		//Переменные для работы с MPX_a2_2
	mpx_a2_2_in_v_1 	 		   		:WORD; //1-е Напрядение входа
	mpx_a2_2_in_v_2 	 		   		:WORD; //2-e Напряжение входа
	mpx_a2_2_in_v_3 	 		   		:WORD; //3-е Напряжение входа
	mpx_a2_2_in_freq 	 		   		:WORD; //Частота на входе
	mpx_a2_2_in_freq_real		   		:REAL; //Частота на входе (x0.1)
	mpx_a2_2_bypass_v_1  		   		:WORD; //1-е Напряжение байпаса
	mpx_a2_2_bypass_v_2  		   		:WORD; //2-е Напряжение байпаса
	mpx_a2_2_bypass_v_3  		   		:WORD; //3-е Напряжение байпаса
	mpx_a2_2_bypass_freq 		   		:WORD; //Частота байпаса
	mpx_a2_2_bypass_freq_real      		:REAL; //Частота байпаса
	mpx_a2_2_output_v_1  		   		:WORD; //1-е Напряжение выхода
	mpx_a2_2_output_v_2  		   		:WORD; //2-е Напряжение выхода
	mpx_a2_2_output_v_3  		   		:WORD; //3-е Напряжение выхода
	mpx_a2_2_output_i_1  		   		:WORD; //1-й Ток выхода
	mpx_a2_2_output_i_2  		   		:WORD; //2-й Ток выхода
	mpx_a2_2_output_i_3  		   		:WORD; //3-й Ток выхода
	mpx_a2_2_output_i_1_real       		:REAL; //1-й Ток выхода (x0.1)
	mpx_a2_2_output_i_2_real       		:REAL; //2-й Ток выхода (x0.1)
	mpx_a2_2_output_i_3_real       		:REAL; //3-й Ток выхода (x0.1)
	mpx_a2_2_output_active_power_1 		:WORD; //Активная мощность 1-й фазы
	mpx_a2_2_output_active_power_2 		:WORD; //Активная мощность 2-й фазы
	mpx_a2_2_output_active_power_3 		:WORD; //Активная мощность 3-й фазы
	mpx_a2_2_output_active_power_1_real :REAL; //Активная мощность 1-й фазы (x0.1)
	mpx_a2_2_output_active_power_2_real :REAL; //Активная мощность 2-й фазы (x0.1)
	mpx_a2_2_output_active_power_3_real :REAL; //Активная мощность 3-й фазы (x0.1)
	mpx_a2_2_output_freq 	       		:WORD; //Частота выхода
	mpx_a2_2_output_freq_real 	        :REAL; //Частота выхода (x0.1)
	mpx_a2_2_load_ph_1    	       		:WORD; //Загрузска 1-й фазы (%)
	mpx_a2_2_load_ph_2    		   		:WORD; //Загрузска 3-й фазы (%)
	mpx_a2_2_load_ph_3    	       		:WORD; //Загрузска 2-й фазы (%)
	mpx_a2_2_battery_voltage 	   		:WORD; //Напряжение батареи
	mpx_a2_2_battery_voltage_real  		:REAL; //Напряжение батареи (x0.1)
	mpx_a2_2_battery_current 	   		:WORD; //Ток батареи
	mpx_a2_2_battery_current_real  		:REAL; //Ток батареи (x0.1)
	mpx_a2_2_battery_capacity 	   		:WORD; //Остаточная емкость батареи (%)
	mpx_a2_2_battery_time 		   		:WORD; //Остаточное время автономии (минуты)
	mpx_a2_2_temp 				   		:WORD; //Температура
	mpx_a2_2_state_reg_1 	       		:WORD; //1-й Регистр состояния
	mpx_a2_2_state_1_as_bit 	   		:WORD_AS_BIT;
	mpx_a2_2_state_reg_2 		   		:WORD; //2-й Регистр состояния
	mpx_a2_2_state_2_as_bit 	   		:WORD_AS_BIT;
	mpx_a2_2_bypass_line_state 	   		:STRING; 
	mpx_a2_2_bypass_arrow_state    		:STRING;
	mpx_a2_2_battery_arrow_state 		:STRING; //состояние батареи
	mpx_a2_2_battery_line_state 		:STRING; //состояние батареи
	mpx_a2_2_input_state 		   		:STRING; //состояние входа
	mpx_a2_2_output_state 		   		:STRING; //состояние выхода
	mpx_a2_2_alarm                      :BOOL;
	
	//Переменные для работы с MPX_s1_1
	mpx_s1_1_in_v_1 	 		   		:WORD; //1-е Напрядение входа
	mpx_s1_1_in_v_2 	 		   		:WORD; //2-e Напряжение входа
	mpx_s1_1_in_v_3 	 		   		:WORD; //3-е Напряжение входа
	mpx_s1_1_in_freq 	 		   		:WORD; //Частота на входе
	mpx_s1_1_in_freq_real		   		:REAL; //Частота на входе (x0.1)
	mpx_s1_1_bypass_v_1  		   		:WORD; //1-е Напряжение байпаса
	mpx_s1_1_bypass_v_2  		   		:WORD; //2-е Напряжение байпаса
	mpx_s1_1_bypass_v_3  		   		:WORD; //3-е Напряжение байпаса
	mpx_s1_1_bypass_freq 		   		:WORD; //Частота байпаса
	mpx_s1_1_bypass_freq_real      		:REAL; //Частота байпаса
	mpx_s1_1_output_v_1  		   		:WORD; //1-е Напряжение выхода
	mpx_s1_1_output_v_2  		   		:WORD; //2-е Напряжение выхода
	mpx_s1_1_output_v_3  		   		:WORD; //3-е Напряжение выхода
	mpx_s1_1_output_i_1  		   		:WORD; //1-й Ток выхода
	mpx_s1_1_output_i_2  		   		:WORD; //2-й Ток выхода
	mpx_s1_1_output_i_3  		   		:WORD; //3-й Ток выхода
	mpx_s1_1_output_i_1_real       		:REAL; //1-й Ток выхода (x0.1)
	mpx_s1_1_output_i_2_real       		:REAL; //2-й Ток выхода (x0.1)
	mpx_s1_1_output_i_3_real       		:REAL; //3-й Ток выхода (x0.1)
	mpx_s1_1_output_active_power_1 		:WORD; //Активная мощность 1-й фазы
	mpx_s1_1_output_active_power_2 		:WORD; //Активная мощность 2-й фазы
	mpx_s1_1_output_active_power_3 		:WORD; //Активная мощность 3-й фазы
	mpx_s1_1_output_active_power_1_real :REAL; //Активная мощность 1-й фазы (x0.1)
	mpx_s1_1_output_active_power_2_real :REAL; //Активная мощность 2-й фазы (x0.1)
	mpx_s1_1_output_active_power_3_real :REAL; //Активная мощность 3-й фазы (x0.1)
	mpx_s1_1_output_freq 	       		:WORD; //Частота выхода
	mpx_s1_1_output_freq_real 	        :REAL; //Частота выхода (x0.1)
	mpx_s1_1_load_ph_1    	       		:WORD; //Загрузска 1-й фазы (%)
	mpx_s1_1_load_ph_2    		   		:WORD; //Загрузска 3-й фазы (%)
	mpx_s1_1_load_ph_3    	       		:WORD; //Загрузска 2-й фазы (%)
	mpx_s1_1_battery_voltage 	   		:WORD; //Напряжение батареи
	mpx_s1_1_battery_voltage_real  		:REAL; //Напряжение батареи (x0.1)
	mpx_s1_1_battery_current 	   		:WORD; //Ток батареи
	mpx_s1_1_battery_current_real  		:REAL; //Ток батареи (x0.1)
	mpx_s1_1_battery_capacity 	   		:WORD; //Остаточная емкость батареи (%)
	mpx_s1_1_battery_time 		   		:WORD; //Остаточное время автономии (минуты)
	mpx_s1_1_temp 				   		:WORD; //Температура
	mpx_s1_1_state_reg_1 	       		:WORD; //1-й Регистр состояния
	mpx_s1_1_state_1_as_bit 	   		:WORD_AS_BIT;
	mpx_s1_1_state_reg_2 		   		:WORD; //2-й Регистр состояния
	mpx_s1_1_state_2_as_bit 	   		:WORD_AS_BIT;
	mpx_s1_1_bypass_line_state 	   		:STRING; 
	mpx_s1_1_bypass_arrow_state    		:STRING;
	mpx_s1_1_battery_arrow_state 		:STRING; //состояние батареи
	mpx_s1_1_battery_line_state 		:STRING; //состояние батареи
	mpx_s1_1_input_state 		   		:STRING; //состояние входа
	mpx_s1_1_output_state 		   		:STRING; //состояние выхода
	mpx_s1_1_alarm                      :BOOL;
	
	//Переменные для работы с MPX_s1_2
	mpx_s1_2_in_v_1 	 		   		:WORD; //1-е Напрядение входа
	mpx_s1_2_in_v_2 	 		   		:WORD; //2-e Напряжение входа
	mpx_s1_2_in_v_3 	 		   		:WORD; //3-е Напряжение входа
	mpx_s1_2_in_freq 	 		   		:WORD; //Частота на входе
	mpx_s1_2_in_freq_real		   		:REAL; //Частота на входе (x0.1)
	mpx_s1_2_bypass_v_1  		   		:WORD; //1-е Напряжение байпаса
	mpx_s1_2_bypass_v_2  		   		:WORD; //2-е Напряжение байпаса
	mpx_s1_2_bypass_v_3  		   		:WORD; //3-е Напряжение байпаса
	mpx_s1_2_bypass_freq 		   		:WORD; //Частота байпаса
	mpx_s1_2_bypass_freq_real      		:REAL; //Частота байпаса
	mpx_s1_2_output_v_1  		   		:WORD; //1-е Напряжение выхода
	mpx_s1_2_output_v_2  		   		:WORD; //2-е Напряжение выхода
	mpx_s1_2_output_v_3  		   		:WORD; //3-е Напряжение выхода
	mpx_s1_2_output_i_1  		   		:WORD; //1-й Ток выхода
	mpx_s1_2_output_i_2  		   		:WORD; //2-й Ток выхода
	mpx_s1_2_output_i_3  		   		:WORD; //3-й Ток выхода
	mpx_s1_2_output_i_1_real       		:REAL; //1-й Ток выхода (x0.1)
	mpx_s1_2_output_i_2_real       		:REAL; //2-й Ток выхода (x0.1)
	mpx_s1_2_output_i_3_real       		:REAL; //3-й Ток выхода (x0.1)
	mpx_s1_2_output_active_power_1 		:WORD; //Активная мощность 1-й фазы
	mpx_s1_2_output_active_power_2 		:WORD; //Активная мощность 2-й фазы
	mpx_s1_2_output_active_power_3 		:WORD; //Активная мощность 3-й фазы
	mpx_s1_2_output_active_power_1_real :REAL; //Активная мощность 1-й фазы (x0.1)
	mpx_s1_2_output_active_power_2_real :REAL; //Активная мощность 2-й фазы (x0.1)
	mpx_s1_2_output_active_power_3_real :REAL; //Активная мощность 3-й фазы (x0.1)
	mpx_s1_2_output_freq 	       		:WORD; //Частота выхода
	mpx_s1_2_output_freq_real 	        :REAL; //Частота выхода (x0.1)
	mpx_s1_2_load_ph_1    	       		:WORD; //Загрузска 1-й фазы (%)
	mpx_s1_2_load_ph_2    		   		:WORD; //Загрузска 3-й фазы (%)
	mpx_s1_2_load_ph_3    	       		:WORD; //Загрузска 2-й фазы (%)
	mpx_s1_2_battery_voltage 	   		:WORD; //Напряжение батареи
	mpx_s1_2_battery_voltage_real  		:REAL; //Напряжение батареи (x0.1)
	mpx_s1_2_battery_current 	   		:WORD; //Ток батареи
	mpx_s1_2_battery_current_real  		:REAL; //Ток батареи (x0.1)
	mpx_s1_2_battery_capacity 	   		:WORD; //Остаточная емкость батареи (%)
	mpx_s1_2_battery_time 		   		:WORD; //Остаточное время автономии (минуты)
	mpx_s1_2_temp 				   		:WORD; //Температура
	mpx_s1_2_state_reg_1 	       		:WORD; //1-й Регистр состояния
	mpx_s1_2_state_1_as_bit 	   		:WORD_AS_BIT;
	mpx_s1_2_state_reg_2 		   		:WORD; //2-й Регистр состояния
	mpx_s1_2_state_2_as_bit 	   		:WORD_AS_BIT;
	mpx_s1_2_bypass_line_state 	   		:STRING; 
	mpx_s1_2_bypass_arrow_state    		:STRING;
	mpx_s1_2_battery_arrow_state 		:STRING; //состояние батареи
	mpx_s1_2_battery_line_state 		:STRING; //состояние батареи
	mpx_s1_2_input_state 		   		:STRING; //состояние входа
	mpx_s1_2_output_state 		   		:STRING; //состояние выхода
	mpx_s1_2_alarm                      :BOOL;
	
	//Переменные для работы с MPX_s1_3
	mpx_s1_3_in_v_1 	 		   		:WORD; //1-е Напрядение входа
	mpx_s1_3_in_v_2 	 		   		:WORD; //2-e Напряжение входа
	mpx_s1_3_in_v_3 	 		   		:WORD; //3-е Напряжение входа
	mpx_s1_3_in_freq 	 		   		:WORD; //Частота на входе
	mpx_s1_3_in_freq_real		   		:REAL; //Частота на входе (x0.1)
	mpx_s1_3_bypass_v_1  		   		:WORD; //1-е Напряжение байпаса
	mpx_s1_3_bypass_v_2  		   		:WORD; //2-е Напряжение байпаса
	mpx_s1_3_bypass_v_3  		   		:WORD; //3-е Напряжение байпаса
	mpx_s1_3_bypass_freq 		   		:WORD; //Частота байпаса
	mpx_s1_3_bypass_freq_real      		:REAL; //Частота байпаса
	mpx_s1_3_output_v_1  		   		:WORD; //1-е Напряжение выхода
	mpx_s1_3_output_v_2  		   		:WORD; //2-е Напряжение выхода
	mpx_s1_3_output_v_3  		   		:WORD; //3-е Напряжение выхода
	mpx_s1_3_output_i_1  		   		:WORD; //1-й Ток выхода
	mpx_s1_3_output_i_2  		   		:WORD; //2-й Ток выхода
	mpx_s1_3_output_i_3  		   		:WORD; //3-й Ток выхода
	mpx_s1_3_output_i_1_real       		:REAL; //1-й Ток выхода (x0.1)
	mpx_s1_3_output_i_2_real       		:REAL; //2-й Ток выхода (x0.1)
	mpx_s1_3_output_i_3_real       		:REAL; //3-й Ток выхода (x0.1)
	mpx_s1_3_output_active_power_1 		:WORD; //Активная мощность 1-й фазы
	mpx_s1_3_output_active_power_2 		:WORD; //Активная мощность 2-й фазы
	mpx_s1_3_output_active_power_3 		:WORD; //Активная мощность 3-й фазы
	mpx_s1_3_output_active_power_1_real :REAL; //Активная мощность 1-й фазы (x0.1)
	mpx_s1_3_output_active_power_2_real :REAL; //Активная мощность 2-й фазы (x0.1)
	mpx_s1_3_output_active_power_3_real :REAL; //Активная мощность 3-й фазы (x0.1)
	mpx_s1_3_output_freq 	       		:WORD; //Частота выхода
	mpx_s1_3_output_freq_real 	        :REAL; //Частота выхода (x0.1)
	mpx_s1_3_load_ph_1    	       		:WORD; //Загрузска 1-й фазы (%)
	mpx_s1_3_load_ph_2    		   		:WORD; //Загрузска 3-й фазы (%)
	mpx_s1_3_load_ph_3    	       		:WORD; //Загрузска 2-й фазы (%)
	mpx_s1_3_battery_voltage 	   		:WORD; //Напряжение батареи
	mpx_s1_3_battery_voltage_real  		:REAL; //Напряжение батареи (x0.1)
	mpx_s1_3_battery_current 	   		:WORD; //Ток батареи
	mpx_s1_3_battery_current_real  		:REAL; //Ток батареи (x0.1)
	mpx_s1_3_battery_capacity 	   		:WORD; //Остаточная емкость батареи (%)
	mpx_s1_3_battery_time 		   		:WORD; //Остаточное время автономии (минуты)
	mpx_s1_3_temp 				   		:WORD; //Температура
	mpx_s1_3_state_reg_1 	       		:WORD; //1-й Регистр состояния
	mpx_s1_3_state_1_as_bit 	   		:WORD_AS_BIT;
	mpx_s1_3_state_reg_2 		   		:WORD; //2-й Регистр состояния
	mpx_s1_3_state_2_as_bit 	   		:WORD_AS_BIT;
	mpx_s1_3_bypass_line_state 	   		:STRING; 
	mpx_s1_3_bypass_arrow_state    		:STRING;
	mpx_s1_3_battery_arrow_state 		:STRING; //состояние батареи
	mpx_s1_3_battery_line_state 		:STRING; //состояние батареи
	mpx_s1_3_input_state 		   		:STRING; //состояние входа
	mpx_s1_3_output_state 		   		:STRING; //состояние выхода
	mpx_s1_3_alarm                      :BOOL;
	
	//Переменные для работы с MPX_s1_4
	mpx_s1_4_in_v_1 	 		   		:WORD; //1-е Напрядение входа
	mpx_s1_4_in_v_2 	 		   		:WORD; //2-e Напряжение входа
	mpx_s1_4_in_v_3 	 		   		:WORD; //3-е Напряжение входа
	mpx_s1_4_in_freq 	 		   		:WORD; //Частота на входе
	mpx_s1_4_in_freq_real		   		:REAL; //Частота на входе (x0.1)
	mpx_s1_4_bypass_v_1  		   		:WORD; //1-е Напряжение байпаса
	mpx_s1_4_bypass_v_2  		   		:WORD; //2-е Напряжение байпаса
	mpx_s1_4_bypass_v_3  		   		:WORD; //3-е Напряжение байпаса
	mpx_s1_4_bypass_freq 		   		:WORD; //Частота байпаса
	mpx_s1_4_bypass_freq_real      		:REAL; //Частота байпаса
	mpx_s1_4_output_v_1  		   		:WORD; //1-е Напряжение выхода
	mpx_s1_4_output_v_2  		   		:WORD; //2-е Напряжение выхода
	mpx_s1_4_output_v_3  		   		:WORD; //3-е Напряжение выхода
	mpx_s1_4_output_i_1  		   		:WORD; //1-й Ток выхода
	mpx_s1_4_output_i_2  		   		:WORD; //2-й Ток выхода
	mpx_s1_4_output_i_3  		   		:WORD; //3-й Ток выхода
	mpx_s1_4_output_i_1_real       		:REAL; //1-й Ток выхода (x0.1)
	mpx_s1_4_output_i_2_real       		:REAL; //2-й Ток выхода (x0.1)
	mpx_s1_4_output_i_3_real       		:REAL; //3-й Ток выхода (x0.1)
	mpx_s1_4_output_active_power_1 		:WORD; //Активная мощность 1-й фазы
	mpx_s1_4_output_active_power_2 		:WORD; //Активная мощность 2-й фазы
	mpx_s1_4_output_active_power_3 		:WORD; //Активная мощность 3-й фазы
	mpx_s1_4_output_active_power_1_real :REAL; //Активная мощность 1-й фазы (x0.1)
	mpx_s1_4_output_active_power_2_real :REAL; //Активная мощность 2-й фазы (x0.1)
	mpx_s1_4_output_active_power_3_real :REAL; //Активная мощность 3-й фазы (x0.1)
	mpx_s1_4_output_freq 	       		:WORD; //Частота выхода
	mpx_s1_4_output_freq_real 	        :REAL; //Частота выхода (x0.1)
	mpx_s1_4_load_ph_1    	       		:WORD; //Загрузска 1-й фазы (%)
	mpx_s1_4_load_ph_2    		   		:WORD; //Загрузска 3-й фазы (%)
	mpx_s1_4_load_ph_3    	       		:WORD; //Загрузска 2-й фазы (%)
	mpx_s1_4_battery_voltage 	   		:WORD; //Напряжение батареи
	mpx_s1_4_battery_voltage_real  		:REAL; //Напряжение батареи (x0.1)
	mpx_s1_4_battery_current 	   		:WORD; //Ток батареи
	mpx_s1_4_battery_current_real  		:REAL; //Ток батареи (x0.1)
	mpx_s1_4_battery_capacity 	   		:WORD; //Остаточная емкость батареи (%)
	mpx_s1_4_battery_time 		   		:WORD; //Остаточное время автономии (минуты)
	mpx_s1_4_temp 				   		:WORD; //Температура
	mpx_s1_4_state_reg_1 	       		:WORD; //1-й Регистр состояния
	mpx_s1_4_state_1_as_bit 	   		:WORD_AS_BIT;
	mpx_s1_4_state_reg_2 		   		:WORD; //2-й Регистр состояния
	mpx_s1_4_state_2_as_bit 	   		:WORD_AS_BIT;
	mpx_s1_4_bypass_line_state 	   		:STRING; 
	mpx_s1_4_bypass_arrow_state    		:STRING;
	mpx_s1_4_battery_arrow_state 		:STRING; //состояние батареи
	mpx_s1_4_battery_line_state 		:STRING; //состояние батареи
	mpx_s1_4_input_state 		   		:STRING; //состояние входа
	mpx_s1_4_output_state 		   		:STRING; //состояние выхода
	mpx_s1_4_alarm                      :BOOL;
	
	//Переменные для работы с MPX_s2_1
	mpx_s2_1_in_v_1 	 		   		:WORD; //1-е Напрядение входа
	mpx_s2_1_in_v_2 	 		   		:WORD; //2-e Напряжение входа
	mpx_s2_1_in_v_3 	 		   		:WORD; //3-е Напряжение входа
	mpx_s2_1_in_freq 	 		   		:WORD; //Частота на входе
	mpx_s2_1_in_freq_real		   		:REAL; //Частота на входе (x0.1)
	mpx_s2_1_bypass_v_1  		   		:WORD; //1-е Напряжение байпаса
	mpx_s2_1_bypass_v_2  		   		:WORD; //2-е Напряжение байпаса
	mpx_s2_1_bypass_v_3  		   		:WORD; //3-е Напряжение байпаса
	mpx_s2_1_bypass_freq 		   		:WORD; //Частота байпаса
	mpx_s2_1_bypass_freq_real      		:REAL; //Частота байпаса
	mpx_s2_1_output_v_1  		   		:WORD; //1-е Напряжение выхода
	mpx_s2_1_output_v_2  		   		:WORD; //2-е Напряжение выхода
	mpx_s2_1_output_v_3  		   		:WORD; //3-е Напряжение выхода
	mpx_s2_1_output_i_1  		   		:WORD; //1-й Ток выхода
	mpx_s2_1_output_i_2  		   		:WORD; //2-й Ток выхода
	mpx_s2_1_output_i_3  		   		:WORD; //3-й Ток выхода
	mpx_s2_1_output_i_1_real       		:REAL; //1-й Ток выхода (x0.1)
	mpx_s2_1_output_i_2_real       		:REAL; //2-й Ток выхода (x0.1)
	mpx_s2_1_output_i_3_real       		:REAL; //3-й Ток выхода (x0.1)
	mpx_s2_1_output_active_power_1 		:WORD; //Активная мощность 1-й фазы
	mpx_s2_1_output_active_power_2 		:WORD; //Активная мощность 2-й фазы
	mpx_s2_1_output_active_power_3 		:WORD; //Активная мощность 3-й фазы
	mpx_s2_1_output_active_power_1_real :REAL; //Активная мощность 1-й фазы (x0.1)
	mpx_s2_1_output_active_power_2_real :REAL; //Активная мощность 2-й фазы (x0.1)
	mpx_s2_1_output_active_power_3_real :REAL; //Активная мощность 3-й фазы (x0.1)
	mpx_s2_1_output_freq 	       		:WORD; //Частота выхода
	mpx_s2_1_output_freq_real 	        :REAL; //Частота выхода (x0.1)
	mpx_s2_1_load_ph_1    	       		:WORD; //Загрузска 1-й фазы (%)
	mpx_s2_1_load_ph_2    		   		:WORD; //Загрузска 3-й фазы (%)
	mpx_s2_1_load_ph_3    	       		:WORD; //Загрузска 2-й фазы (%)
	mpx_s2_1_battery_voltage 	   		:WORD; //Напряжение батареи
	mpx_s2_1_battery_voltage_real  		:REAL; //Напряжение батареи (x0.1)
	mpx_s2_1_battery_current 	   		:WORD; //Ток батареи
	mpx_s2_1_battery_current_real  		:REAL; //Ток батареи (x0.1)
	mpx_s2_1_battery_capacity 	   		:WORD; //Остаточная емкость батареи (%)
	mpx_s2_1_battery_time 		   		:WORD; //Остаточное время автономии (минуты)
	mpx_s2_1_temp 				   		:WORD; //Температура
	mpx_s2_1_state_reg_1 	       		:WORD; //1-й Регистр состояния
	mpx_s2_1_state_1_as_bit 	   		:WORD_AS_BIT;
	mpx_s2_1_state_reg_2 		   		:WORD; //2-й Регистр состояния
	mpx_s2_1_state_2_as_bit 	   		:WORD_AS_BIT;
	mpx_s2_1_bypass_line_state 	   		:STRING; 
	mpx_s2_1_bypass_arrow_state    		:STRING;
	mpx_s2_1_battery_arrow_state 		:STRING; //состояние батареи
	mpx_s2_1_battery_line_state 		:STRING; //состояние батареи
	mpx_s2_1_input_state 		   		:STRING; //состояние входа
	mpx_s2_1_output_state 		   		:STRING; //состояние выхода
	mpx_s2_1_alarm                      :BOOL;

	//Переменные для работы с MPX_S2_2
	mpx_s2_2_in_v_1 	 		   		:WORD; //1-е Напрядение входа
	mpx_s2_2_in_v_2 	 		   		:WORD; //2-e Напряжение входа
	mpx_s2_2_in_v_3 	 		   		:WORD; //3-е Напряжение входа
	mpx_s2_2_in_freq 	 		   		:WORD; //Частота на входе
	mpx_s2_2_in_freq_real		   		:REAL; //Частота на входе (x0.1)
	mpx_s2_2_bypass_v_1  		   		:WORD; //1-е Напряжение байпаса
	mpx_s2_2_bypass_v_2  		   		:WORD; //2-е Напряжение байпаса
	mpx_s2_2_bypass_v_3  		   		:WORD; //3-е Напряжение байпаса
	mpx_s2_2_bypass_freq 		   		:WORD; //Частота байпаса
	mpx_s2_2_bypass_freq_real      		:REAL; //Частота байпаса
	mpx_s2_2_output_v_1  		   		:WORD; //1-е Напряжение выхода
	mpx_s2_2_output_v_2  		   		:WORD; //2-е Напряжение выхода
	mpx_s2_2_output_v_3  		   		:WORD; //3-е Напряжение выхода
	mpx_s2_2_output_i_1  		   		:WORD; //1-й Ток выхода
	mpx_s2_2_output_i_2  		   		:WORD; //2-й Ток выхода
	mpx_s2_2_output_i_3  		   		:WORD; //3-й Ток выхода
	mpx_s2_2_output_i_1_real       		:REAL; //1-й Ток выхода (x0.1)
	mpx_s2_2_output_i_2_real       		:REAL; //2-й Ток выхода (x0.1)
	mpx_s2_2_output_i_3_real       		:REAL; //3-й Ток выхода (x0.1)
	mpx_s2_2_output_active_power_1 		:WORD; //Активная мощность 1-й фазы
	mpx_s2_2_output_active_power_2 		:WORD; //Активная мощность 2-й фазы
	mpx_s2_2_output_active_power_3 		:WORD; //Активная мощность 3-й фазы
	mpx_s2_2_output_active_power_1_real :REAL; //Активная мощность 1-й фазы (x0.1)
	mpx_s2_2_output_active_power_2_real :REAL; //Активная мощность 2-й фазы (x0.1)
	mpx_s2_2_output_active_power_3_real :REAL; //Активная мощность 3-й фазы (x0.1)
	mpx_s2_2_output_freq 	       		:WORD; //Частота выхода
	mpx_s2_2_output_freq_real 	        :REAL; //Частота выхода (x0.1)
	mpx_s2_2_load_ph_1    	       		:WORD; //Загрузска 1-й фазы (%)
	mpx_s2_2_load_ph_2    		   		:WORD; //Загрузска 3-й фазы (%)
	mpx_s2_2_load_ph_3    	       		:WORD; //Загрузска 2-й фазы (%)
	mpx_s2_2_battery_voltage 	   		:WORD; //Напряжение батареи
	mpx_s2_2_battery_voltage_real  		:REAL; //Напряжение батареи (x0.1)
	mpx_s2_2_battery_current 	   		:WORD; //Ток батареи
	mpx_s2_2_battery_current_real  		:REAL; //Ток батареи (x0.1)
	mpx_s2_2_battery_capacity 	   		:WORD; //Остаточная емкость батареи (%)
	mpx_s2_2_battery_time 		   		:WORD; //Остаточное время автономии (минуты)
	mpx_s2_2_temp 				   		:WORD; //Температура
	mpx_s2_2_state_reg_1 	       		:WORD; //1-й Регистр состояния
	mpx_s2_2_state_1_as_bit 	   		:WORD_AS_BIT;
	mpx_s2_2_state_reg_2 		   		:WORD; //2-й Регистр состояния
	mpx_s2_2_state_2_as_bit 	   		:WORD_AS_BIT;
	mpx_s2_2_bypass_line_state 	   		:STRING; 
	mpx_s2_2_bypass_arrow_state    		:STRING;
	mpx_s2_2_battery_arrow_state 		:STRING; //состояние батареи
	mpx_s2_2_battery_line_state 		:STRING; //состояние батареи
	mpx_s2_2_input_state 		   		:STRING; //состояние входа
	mpx_s2_2_output_state 		   		:STRING; //состояние выхода
	mpx_s2_2_alarm                      :BOOL;
	
	//Переменные для работы с MPX_S2_3
	mpx_s2_3_in_v_1 	 		   		:WORD; //1-е Напрядение входа
	mpx_s2_3_in_v_2 	 		   		:WORD; //2-e Напряжение входа
	mpx_s2_3_in_v_3 	 		   		:WORD; //3-е Напряжение входа
	mpx_s2_3_in_freq 	 		   		:WORD; //Частота на входе
	mpx_s2_3_in_freq_real		   		:REAL; //Частота на входе (x0.1)
	mpx_s2_3_bypass_v_1  		   		:WORD; //1-е Напряжение байпаса
	mpx_s2_3_bypass_v_2  		   		:WORD; //2-е Напряжение байпаса
	mpx_s2_3_bypass_v_3  		   		:WORD; //3-е Напряжение байпаса
	mpx_s2_3_bypass_freq 		   		:WORD; //Частота байпаса
	mpx_s2_3_bypass_freq_real      		:REAL; //Частота байпаса
	mpx_s2_3_output_v_1  		   		:WORD; //1-е Напряжение выхода
	mpx_s2_3_output_v_2  		   		:WORD; //2-е Напряжение выхода
	mpx_s2_3_output_v_3  		   		:WORD; //3-е Напряжение выхода
	mpx_s2_3_output_i_1  		   		:WORD; //1-й Ток выхода
	mpx_s2_3_output_i_2  		   		:WORD; //2-й Ток выхода
	mpx_s2_3_output_i_3  		   		:WORD; //3-й Ток выхода
	mpx_s2_3_output_i_1_real       		:REAL; //1-й Ток выхода (x0.1)
	mpx_s2_3_output_i_2_real       		:REAL; //2-й Ток выхода (x0.1)
	mpx_s2_3_output_i_3_real       		:REAL; //3-й Ток выхода (x0.1)
	mpx_s2_3_output_active_power_1 		:WORD; //Активная мощность 1-й фазы
	mpx_s2_3_output_active_power_2 		:WORD; //Активная мощность 2-й фазы
	mpx_s2_3_output_active_power_3 		:WORD; //Активная мощность 3-й фазы
	mpx_s2_3_output_active_power_1_real :REAL; //Активная мощность 1-й фазы (x0.1)
	mpx_s2_3_output_active_power_2_real :REAL; //Активная мощность 2-й фазы (x0.1)
	mpx_s2_3_output_active_power_3_real :REAL; //Активная мощность 3-й фазы (x0.1)
	mpx_s2_3_output_freq 	       		:WORD; //Частота выхода
	mpx_s2_3_output_freq_real 	        :REAL; //Частота выхода (x0.1)
	mpx_s2_3_load_ph_1    	       		:WORD; //Загрузска 1-й фазы (%)
	mpx_s2_3_load_ph_2    		   		:WORD; //Загрузска 3-й фазы (%)
	mpx_s2_3_load_ph_3    	       		:WORD; //Загрузска 2-й фазы (%)
	mpx_s2_3_battery_voltage 	   		:WORD; //Напряжение батареи
	mpx_s2_3_battery_voltage_real  		:REAL; //Напряжение батареи (x0.1)
	mpx_s2_3_battery_current 	   		:WORD; //Ток батареи
	mpx_s2_3_battery_current_real  		:REAL; //Ток батареи (x0.1)
	mpx_s2_3_battery_capacity 	   		:WORD; //Остаточная емкость батареи (%)
	mpx_s2_3_battery_time 		   		:WORD; //Остаточное время автономии (минуты)
	mpx_s2_3_temp 				   		:WORD; //Температура
	mpx_s2_3_state_reg_1 	       		:WORD; //1-й Регистр состояния
	mpx_s2_3_state_1_as_bit 	   		:WORD_AS_BIT;
	mpx_s2_3_state_reg_2 		   		:WORD; //2-й Регистр состояния
	mpx_s2_3_state_2_as_bit 	   		:WORD_AS_BIT;
	mpx_s2_3_bypass_line_state 	   		:STRING; 
	mpx_s2_3_bypass_arrow_state    		:STRING;
	mpx_s2_3_battery_arrow_state 		:STRING; //состояние батареи
	mpx_s2_3_battery_line_state 		:STRING; //состояние батареи
	mpx_s2_3_input_state 		   		:STRING; //состояние входа
	mpx_s2_3_output_state 		   		:STRING; //состояние выхода
	mpx_s2_3_alarm                      :BOOL;
	
	//Переменные для работы с MPX_S2_4
	mpx_s2_4_in_v_1 	 		   		:WORD; //1-е Напрядение входа
	mpx_s2_4_in_v_2 	 		   		:WORD; //2-e Напряжение входа
	mpx_s2_4_in_v_3 	 		   		:WORD; //3-е Напряжение входа
	mpx_s2_4_in_freq 	 		   		:WORD; //Частота на входе
	mpx_s2_4_in_freq_real		   		:REAL; //Частота на входе (x0.1)
	mpx_s2_4_bypass_v_1  		   		:WORD; //1-е Напряжение байпаса
	mpx_s2_4_bypass_v_2  		   		:WORD; //2-е Напряжение байпаса
	mpx_s2_4_bypass_v_3  		   		:WORD; //3-е Напряжение байпаса
	mpx_s2_4_bypass_freq 		   		:WORD; //Частота байпаса
	mpx_s2_4_bypass_freq_real      		:REAL; //Частота байпаса
	mpx_s2_4_output_v_1  		   		:WORD; //1-е Напряжение выхода
	mpx_s2_4_output_v_2  		   		:WORD; //2-е Напряжение выхода
	mpx_s2_4_output_v_3  		   		:WORD; //3-е Напряжение выхода
	mpx_s2_4_output_i_1  		   		:WORD; //1-й Ток выхода
	mpx_s2_4_output_i_2  		   		:WORD; //2-й Ток выхода
	mpx_s2_4_output_i_3  		   		:WORD; //3-й Ток выхода
	mpx_s2_4_output_i_1_real       		:REAL; //1-й Ток выхода (x0.1)
	mpx_s2_4_output_i_2_real       		:REAL; //2-й Ток выхода (x0.1)
	mpx_s2_4_output_i_3_real       		:REAL; //3-й Ток выхода (x0.1)
	mpx_s2_4_output_active_power_1 		:WORD; //Активная мощность 1-й фазы
	mpx_s2_4_output_active_power_2 		:WORD; //Активная мощность 2-й фазы
	mpx_s2_4_output_active_power_3 		:WORD; //Активная мощность 3-й фазы
	mpx_s2_4_output_active_power_1_real :REAL; //Активная мощность 1-й фазы (x0.1)
	mpx_s2_4_output_active_power_2_real :REAL; //Активная мощность 2-й фазы (x0.1)
	mpx_s2_4_output_active_power_3_real :REAL; //Активная мощность 3-й фазы (x0.1)
	mpx_s2_4_output_freq 	       		:WORD; //Частота выхода
	mpx_s2_4_output_freq_real 	        :REAL; //Частота выхода (x0.1)
	mpx_s2_4_load_ph_1    	       		:WORD; //Загрузска 1-й фазы (%)
	mpx_s2_4_load_ph_2    		   		:WORD; //Загрузска 3-й фазы (%)
	mpx_s2_4_load_ph_3    	       		:WORD; //Загрузска 2-й фазы (%)
	mpx_s2_4_battery_voltage 	   		:WORD; //Напряжение батареи
	mpx_s2_4_battery_voltage_real  		:REAL; //Напряжение батареи (x0.1)
	mpx_s2_4_battery_current 	   		:WORD; //Ток батареи
	mpx_s2_4_battery_current_real  		:REAL; //Ток батареи (x0.1)
	mpx_s2_4_battery_capacity 	   		:WORD; //Остаточная емкость батареи (%)
	mpx_s2_4_battery_time 		   		:WORD; //Остаточное время автономии (минуты)
	mpx_s2_4_temp 				   		:WORD; //Температура
	mpx_s2_4_state_reg_1 	       		:WORD; //1-й Регистр состояния
	mpx_s2_4_state_1_as_bit 	   		:WORD_AS_BIT;
	mpx_s2_4_state_reg_2 		   		:WORD; //2-й Регистр состояния
	mpx_s2_4_state_2_as_bit 	   		:WORD_AS_BIT;
	mpx_s2_4_bypass_line_state 	   		:STRING; 
	mpx_s2_4_bypass_arrow_state    		:STRING;
	mpx_s2_4_battery_arrow_state 		:STRING; //состояние батареи
	mpx_s2_4_battery_line_state 		:STRING; //состояние батареи
	mpx_s2_4_input_state 		   		:STRING; //состояние входа
	mpx_s2_4_output_state 		   		:STRING; //состояние выхода
	mpx_s2_4_alarm                      :BOOL;
	
	mpx_test_battery_command           :WORD:=20;
	mpx_a1_test_battery_start          :BOOL;
	mpx_a2_test_battery_start          :BOOL;	
	mpx_s1_test_battery_start          :BOOL;
	mpx_s2_test_battery_start          :BOOL;
	
	mpx_s1_all_power                   :REAL;
	mpx_s2_all_power                   :REAL;
	mpx_a1_all_power                   :REAL;
	mpx_a2_all_power                   :REAL;
	
	mpx_s1_state_string :WSTRING := "";
	mpx_s2_state_string :WSTRING := "";
	mpx_a1_state_string :WSTRING := "";
	mpx_a2_state_string :WSTRING := "";
	
	TEST : BOOL;
END_VAR

//Работа с модулем ввода (Адрес = 2)
mv110_reg_as_bit(W := mv110_reg);
mv110_in_0_in_main_present    := mv110_reg_as_bit.B00; //ШАСН - наличие напряжения на основном вводе
mv110_in_1_in_reserve_present := mv110_reg_as_bit.B01; //ШАСН - наличие напряжения на резервном вводе
mv110_in_2_bp_sn_present      := mv110_reg_as_bit.B02; //ШАСН - наличие напряжения на шине БП
mv110_in_3_gp_sn_present      := mv110_reg_as_bit.B03; //ШАСН - наличие напряжения на шине ГП
mv110_in_4_qs1_1position      := mv110_reg_as_bit.B04; //ШАСН - QS1 в 1 положении
mv110_in_5_qs1_2position      := mv110_reg_as_bit.B05; //ШАСН - QS1 во 2 положении
mv110_in_6_heat_on            := mv110_reg_as_bit.B06; //Обогрев ключен
mv110_in_7_gp1_u_fault        := mv110_reg_as_bit.B07; //ЩРПС - ГП1 отключена
mv110_in_8_gp2_u_fault        := mv110_reg_as_bit.B08; //ЩРПС - ГП2 отключена


//Работа с климатом
climate_state_as_bit(W    := climate_state_reg);
climate_zaslonka_state    := climate_state_as_bit.B03;
climate_vent_1_state      := climate_state_as_bit.B00;
climate_vent_2_state      := climate_state_as_bit.B01;
climate_condition_1_state := climate_state_as_bit.B04;
climate_condition_2_state := climate_state_as_bit.B05;
climate_heat_state        := climate_state_as_bit.B02;
climate_heat_door_state   := climate_state_as_bit.B06;
climate_auto_state        := climate_state_as_bit.B07;
climat_temp_out_minus     := climate_state_as_bit.B10;
climat_temp_in_minus      := climate_state_as_bit.B09;
climate_temp_out_real     := climate_temp_out * 0.1;
climate_temp_in_real      := climate_temp_in * 0.1;
IF (climat_temp_out_minus = TRUE) THEN
	climate_temp_out_real := climate_temp_out_real * (-1);
END_IF
IF (climat_temp_in_minus = TRUE) THEN
	climate_temp_in_real := climate_temp_in_real * (-1);
END_IF
IF (climate_temp_in_real > 25) THEN
	climate_temp_excess := TRUE;
	ELSE
		climate_temp_excess := FALSE;
END_IF

//------------------------------------MPX_a1-------------------------------------
//Конвертация параметров MPX_a1_1
mpx_a1_1_in_freq_real               := mpx_a1_1_in_freq * 0.1;
mpx_a1_1_bypass_freq_real           := mpx_a1_1_bypass_freq * 0.1;
mpx_a1_1_output_i_1_real            := mpx_a1_1_output_i_1 * 0.1;
mpx_a1_1_output_active_power_1_real := mpx_a1_1_output_active_power_1 * 0.1;
mpx_a1_1_output_freq_real           := mpx_a1_1_output_freq * 0.1;
mpx_a1_1_battery_voltage_real       := mpx_a1_1_battery_voltage * 0.1;
mpx_a1_1_battery_current_real       := mpx_a1_1_battery_current * 0.1;

//Логика состояний MPX_a1_1
mpx_a1_1_state_1_as_bit(W := mpx_a1_1_state_reg_1);
mpx_a1_1_state_2_as_bit(W := mpx_a1_1_state_reg_2);

IF (mpx_a1_1_state_1_as_bit.B15 = FALSE) THEN
	mpx_a1_1_output_state := 'arrow_off';
	ELSE
		mpx_a1_1_output_state := 'arrow_on';
		mpx_a1_state_string := "От всети";	
END_IF
IF (mpx_a1_1_state_2_as_bit.B12 = FALSE) THEN
	mpx_a1_1_input_state := 'arrow_off';
	ELSE
		mpx_a1_1_input_state := 'arrow_on';	
		mpx_a1_state_string := "От сети";
END_IF
IF (mpx_a1_1_state_1_as_bit.B13 = FALSE) THEN
	mpx_a1_1_battery_line_state := 'battery_line_off';
	mpx_a1_1_battery_arrow_state := 'battery_arrow_off';
	ELSE
		mpx_a1_1_battery_line_state := 'battery_line_on';
		mpx_a1_1_battery_arrow_state := 'battery_arrow_on';	
		mpx_a1_state_string := "От АКБ";
END_IF
IF (mpx_a1_1_state_1_as_bit.B11 = FALSE) THEN
	mpx_a1_1_bypass_line_state := 'bypass_line1_off';
	mpx_a1_1_bypass_arrow_state := 'bypass_arrow_off';
	ELSE
		mpx_a1_1_bypass_line_state := 'bypass_line_on';
		mpx_a1_1_bypass_arrow_state := 'bypass_arrow_on';
		mpx_a1_state_string := "Байпас";	
END_IF
IF ( (mpx_a1_1_state_2_as_bit.B13 = TRUE) OR (mpx_a1_1_state_2_as_bit.B14 = TRUE) OR (mpx_a1_1_state_2_as_bit.B15 = TRUE) ) THEN
	mpx_a1_1_alarm := TRUE;
	ELSE
		mpx_a1_1_alarm := FALSE;
END_IF

//Конвертация параметров MPX_a1_2
mpx_a1_2_in_freq_real               := mpx_a1_2_in_freq * 0.1;
mpx_a1_2_bypass_freq_real           := mpx_a1_2_bypass_freq * 0.1;
mpx_a1_2_output_i_1_real            := mpx_a1_2_output_i_1 * 0.1;
mpx_a1_2_output_active_power_1_real := mpx_a1_2_output_active_power_1 * 0.1;
mpx_a1_2_output_freq_real           := mpx_a1_2_output_freq * 0.1;
mpx_a1_2_battery_voltage_real       := mpx_a1_2_battery_voltage * 0.1;
mpx_a1_2_battery_current_real       := mpx_a1_2_battery_current * 0.1;

//Логика состояний MPX_a1_2
mpx_a1_2_state_1_as_bit(W := mpx_a1_2_state_reg_1);
mpx_a1_2_state_2_as_bit(W := mpx_a1_2_state_reg_2);
IF (mpx_a1_2_state_1_as_bit.B11 = FALSE) THEN
	mpx_a1_2_bypass_line_state := 'bypass_line1_off';
	mpx_a1_2_bypass_arrow_state := 'bypass_arrow_off';
	ELSE
		mpx_a1_2_bypass_line_state := 'bypass_line_on';
		mpx_a1_2_bypass_arrow_state := 'bypass_arrow_on';	
END_IF
IF (mpx_a1_2_state_1_as_bit.B15 = FALSE) THEN
	mpx_a1_2_output_state := 'arrow_off';
	ELSE
		mpx_a1_2_output_state := 'arrow_on';	
END_IF
IF (mpx_a1_2_state_2_as_bit.B12 = FALSE) THEN
	mpx_a1_2_input_state := 'arrow_off';
	ELSE
		mpx_a1_2_input_state := 'arrow_on';	
END_IF
IF (mpx_a1_2_state_1_as_bit.B13 = FALSE) THEN
	mpx_a1_2_battery_line_state := 'battery_line_off';
	mpx_a1_2_battery_arrow_state := 'battery_arrow_off';
	ELSE
		mpx_a1_2_battery_line_state := 'battery_line_on';
		mpx_a1_2_battery_arrow_state := 'battery_arrow_on';	
END_IF
IF ( (mpx_a1_2_state_2_as_bit.B13 = TRUE) OR (mpx_a1_2_state_2_as_bit.B14 = TRUE) OR (mpx_a1_2_state_2_as_bit.B15 = TRUE) ) THEN
	mpx_a1_2_alarm := TRUE;
	ELSE
		mpx_a1_2_alarm := FALSE;
END_IF

mpx_a1_all_power := mpx_a1_2_output_active_power_1_real + mpx_a1_2_output_active_power_1_real;
//------------------------------------MPX_a2-------------------------------------
//Конвертация параметров MPX_a2_1
mpx_a2_1_in_freq_real               := mpx_a2_1_in_freq * 0.1;
mpx_a2_1_bypass_freq_real           := mpx_a2_1_bypass_freq * 0.1;
mpx_a2_1_output_i_1_real            := mpx_a2_1_output_i_1 * 0.1;
mpx_a2_1_output_active_power_1_real := mpx_a2_1_output_active_power_1 * 0.1;
mpx_a2_1_output_freq_real           := mpx_a2_1_output_freq * 0.1;
mpx_a2_1_battery_voltage_real       := mpx_a2_1_battery_voltage * 0.1;
mpx_a2_1_battery_current_real       := mpx_a2_1_battery_current * 0.1;

//Логика состояний MPX_a2_1
mpx_a2_1_state_1_as_bit(W := mpx_a2_1_state_reg_1);
mpx_a2_1_state_2_as_bit(W := mpx_a2_1_state_reg_2);

IF (mpx_a2_1_state_1_as_bit.B15 = FALSE) THEN
	mpx_a2_1_output_state := 'arrow_off';
	ELSE
		mpx_a2_1_output_state := 'arrow_on';
		mpx_a2_state_string := "От всети";	
END_IF
IF (mpx_a2_1_state_2_as_bit.B12 = FALSE) THEN
	mpx_a2_1_input_state := 'arrow_off';
	ELSE
		mpx_a2_1_input_state := 'arrow_on';	
		mpx_a2_state_string := "От сети";
END_IF
IF (mpx_a2_1_state_1_as_bit.B13 = FALSE) THEN
	mpx_a2_1_battery_line_state := 'battery_line_off';
	mpx_a2_1_battery_arrow_state := 'battery_arrow_off';
	ELSE
		mpx_a2_1_battery_line_state := 'battery_line_on';
		mpx_a2_1_battery_arrow_state := 'battery_arrow_on';	
		mpx_a2_state_string := "От АКБ";
END_IF
IF (mpx_a2_1_state_1_as_bit.B11 = FALSE) THEN
	mpx_a2_1_bypass_line_state := 'bypass_line1_off';
	mpx_a2_1_bypass_arrow_state := 'bypass_arrow_off';
	ELSE
		mpx_a2_1_bypass_line_state := 'bypass_line_on';
		mpx_a2_1_bypass_arrow_state := 'bypass_arrow_on';
		mpx_a2_state_string := "Байпас";	
END_IF
IF ( (mpx_a2_1_state_2_as_bit.B13 = TRUE) OR (mpx_a2_1_state_2_as_bit.B14 = TRUE) OR (mpx_a2_1_state_2_as_bit.B15 = TRUE) ) THEN
	mpx_a2_1_alarm := TRUE;
	ELSE
		mpx_a2_1_alarm := FALSE;
END_IF

//Конвертация параметров MPX_a2_2
mpx_a2_2_in_freq_real               := mpx_a2_2_in_freq * 0.1;
mpx_a2_2_bypass_freq_real           := mpx_a2_2_bypass_freq * 0.1;
mpx_a2_2_output_i_1_real            := mpx_a2_2_output_i_1 * 0.1;
mpx_a2_2_output_active_power_1_real := mpx_a2_2_output_active_power_1 * 0.1;
mpx_a2_2_output_freq_real           := mpx_a2_2_output_freq * 0.1;
mpx_a2_2_battery_voltage_real       := mpx_a2_2_battery_voltage * 0.1;
mpx_a2_2_battery_current_real       := mpx_a2_2_battery_current * 0.1;

//Логика состояний MPX_a2_2
mpx_a2_2_state_1_as_bit(W := mpx_a2_2_state_reg_1);
mpx_a2_2_state_2_as_bit(W := mpx_a2_2_state_reg_2);
IF (mpx_a2_2_state_1_as_bit.B11 = FALSE) THEN
	mpx_a2_2_bypass_line_state := 'bypass_line1_off';
	mpx_a2_2_bypass_arrow_state := 'bypass_arrow_off';
	ELSE
		mpx_a2_2_bypass_line_state := 'bypass_line_on';
		mpx_a2_2_bypass_arrow_state := 'bypass_arrow_on';	
END_IF
IF (mpx_a2_2_state_1_as_bit.B15 = FALSE) THEN
	mpx_a2_2_output_state := 'arrow_off';
	ELSE
		mpx_a2_2_output_state := 'arrow_on';	
END_IF
IF (mpx_a2_2_state_2_as_bit.B12 = FALSE) THEN
	mpx_a2_2_input_state := 'arrow_off';
	ELSE
		mpx_a2_2_input_state := 'arrow_on';	
END_IF
IF (mpx_a2_2_state_1_as_bit.B13 = FALSE) THEN
	mpx_a2_2_battery_line_state := 'battery_line_off';
	mpx_a2_2_battery_arrow_state := 'battery_arrow_off';
	ELSE
		mpx_a2_2_battery_line_state := 'battery_line_on';
		mpx_a2_2_battery_arrow_state := 'battery_arrow_on';	
END_IF
IF ( (mpx_a2_2_state_2_as_bit.B13 = TRUE) OR (mpx_a2_2_state_2_as_bit.B14 = TRUE) OR (mpx_a2_2_state_2_as_bit.B15 = TRUE) ) THEN
	mpx_a2_2_alarm := TRUE;
	ELSE
		mpx_a2_2_alarm := FALSE;
END_IF

mpx_a2_all_power := mpx_a2_2_output_active_power_1_real + mpx_a2_2_output_active_power_1_real;
//------------------------------------MPX_S1-------------------------------------
//Конвертация параметров MPX_s1_1
mpx_s1_1_in_freq_real               := mpx_s1_1_in_freq * 0.1;
mpx_s1_1_bypass_freq_real           := mpx_s1_1_bypass_freq * 0.1;
mpx_s1_1_output_i_1_real            := mpx_s1_1_output_i_1 * 0.1;
mpx_s1_1_output_i_2_real            := mpx_s1_1_output_i_2 * 0.1;
mpx_s1_1_output_i_3_real            := mpx_s1_1_output_i_3 * 0.1;
mpx_s1_1_output_active_power_1_real := mpx_s1_1_output_active_power_1 * 0.1;
mpx_s1_1_output_active_power_2_real := mpx_s1_1_output_active_power_2 * 0.1;
mpx_s1_1_output_active_power_3_real := mpx_s1_1_output_active_power_3 * 0.1;
mpx_s1_1_output_freq_real           := mpx_s1_1_output_freq * 0.1;
mpx_s1_1_battery_voltage_real       := mpx_s1_1_battery_voltage * 0.1;
mpx_s1_1_battery_current_real       := mpx_s1_1_battery_current * 0.1;

//Логика состояний MPX_s1_1
mpx_s1_1_state_1_as_bit(W := mpx_s1_1_state_reg_1);
mpx_s1_1_state_2_as_bit(W := mpx_s1_1_state_reg_2);

IF (mpx_s1_1_state_1_as_bit.B15 = FALSE) THEN
	mpx_s1_1_output_state := 'arrow_off';
	ELSE
		mpx_s1_1_output_state := 'arrow_on';
		mpx_s1_state_string := "От всети";	
END_IF
IF (mpx_s1_1_state_2_as_bit.B12 = FALSE) THEN
	mpx_s1_1_input_state := 'arrow_off';
	ELSE
		mpx_s1_1_input_state := 'arrow_on';	
		mpx_s1_state_string := "От сети";
END_IF
IF (mpx_s1_1_state_1_as_bit.B13 = FALSE) THEN
	mpx_s1_1_battery_line_state := 'battery_line_off';
	mpx_s1_1_battery_arrow_state := 'battery_arrow_off';
	ELSE
		mpx_s1_1_battery_line_state := 'battery_line_on';
		mpx_s1_1_battery_arrow_state := 'battery_arrow_on';	
		mpx_s1_state_string := "От АКБ";
END_IF
IF (mpx_s1_1_state_1_as_bit.B11 = FALSE) THEN
	mpx_s1_1_bypass_line_state := 'bypass_line1_off';
	mpx_s1_1_bypass_arrow_state := 'bypass_arrow_off';
	ELSE
		mpx_s1_1_bypass_line_state := 'bypass_line_on';
		mpx_s1_1_bypass_arrow_state := 'bypass_arrow_on';
		mpx_s1_state_string := "Байпас";	
END_IF
IF ( (mpx_s1_1_state_2_as_bit.B13 = TRUE) OR (mpx_s1_1_state_2_as_bit.B14 = TRUE) OR (mpx_s1_1_state_2_as_bit.B15 = TRUE) ) THEN
	mpx_s1_1_alarm := TRUE;
	ELSE
		mpx_s1_1_alarm := FALSE;
END_IF

//Конвертация параметров MPX_s1_2
mpx_s1_2_in_freq_real               := mpx_s1_2_in_freq * 0.1;
mpx_s1_2_bypass_freq_real           := mpx_s1_2_bypass_freq * 0.1;
mpx_s1_2_output_i_1_real            := mpx_s1_2_output_i_1 * 0.1;
mpx_s1_2_output_i_2_real            := mpx_s1_2_output_i_2 * 0.1;
mpx_s1_2_output_i_3_real            := mpx_s1_2_output_i_3 * 0.1;
mpx_s1_2_output_active_power_1_real := mpx_s1_2_output_active_power_1 * 0.1;
mpx_s1_2_output_active_power_2_real := mpx_s1_2_output_active_power_2 * 0.1;
mpx_s1_2_output_active_power_3_real := mpx_s1_2_output_active_power_3 * 0.1;
mpx_s1_2_output_freq_real           := mpx_s1_2_output_freq * 0.1;
mpx_s1_2_battery_voltage_real       := mpx_s1_2_battery_voltage * 0.1;
mpx_s1_2_battery_current_real       := mpx_s1_2_battery_current * 0.1;

//Логика состояний MPX_s1_2
mpx_s1_2_state_1_as_bit(W := mpx_s1_2_state_reg_1);
mpx_s1_2_state_2_as_bit(W := mpx_s1_2_state_reg_2);
IF (mpx_s1_2_state_1_as_bit.B11 = FALSE) THEN
	mpx_s1_2_bypass_line_state := 'bypass_line1_off';
	mpx_s1_2_bypass_arrow_state := 'bypass_arrow_off';
	ELSE
		mpx_s1_2_bypass_line_state := 'bypass_line_on';
		mpx_s1_2_bypass_arrow_state := 'bypass_arrow_on';	
END_IF
IF (mpx_s1_2_state_1_as_bit.B15 = FALSE) THEN
	mpx_s1_2_output_state := 'arrow_off';
	ELSE
		mpx_s1_2_output_state := 'arrow_on';	
END_IF
IF (mpx_s1_2_state_2_as_bit.B12 = FALSE) THEN
	mpx_s1_2_input_state := 'arrow_off';
	ELSE
		mpx_s1_2_input_state := 'arrow_on';	
END_IF
IF (mpx_s1_2_state_1_as_bit.B13 = FALSE) THEN
	mpx_s1_2_battery_line_state := 'battery_line_off';
	mpx_s1_2_battery_arrow_state := 'battery_arrow_off';
	ELSE
		mpx_s1_2_battery_line_state := 'battery_line_on';
		mpx_s1_2_battery_arrow_state := 'battery_arrow_on';	
END_IF
IF ( (mpx_s1_2_state_2_as_bit.B13 = TRUE) OR (mpx_s1_2_state_2_as_bit.B14 = TRUE) OR (mpx_s1_2_state_2_as_bit.B15 = TRUE) ) THEN
	mpx_s1_2_alarm := TRUE;
	ELSE
		mpx_s1_2_alarm := FALSE;
END_IF

//Конвертация параметров MPX_s1_3
mpx_s1_3_in_freq_real               := mpx_s1_3_in_freq * 0.1;
mpx_s1_3_bypass_freq_real           := mpx_s1_3_bypass_freq * 0.1;
mpx_s1_3_output_i_1_real            := mpx_s1_3_output_i_1 * 0.1;
mpx_s1_3_output_i_2_real            := mpx_s1_3_output_i_2 * 0.1;
mpx_s1_3_output_i_3_real            := mpx_s1_3_output_i_3 * 0.1;
mpx_s1_3_output_active_power_1_real := mpx_s1_3_output_active_power_1 * 0.1;
mpx_s1_3_output_active_power_2_real := mpx_s1_3_output_active_power_2 * 0.1;
mpx_s1_3_output_active_power_3_real := mpx_s1_3_output_active_power_3 * 0.1;
mpx_s1_3_output_freq_real           := mpx_s1_3_output_freq * 0.1;
mpx_s1_3_battery_voltage_real       := mpx_s1_3_battery_voltage * 0.1;
mpx_s1_3_battery_current_real       := mpx_s1_3_battery_current * 0.1;

//Логика состояний MPX_s1_3
mpx_s1_3_state_1_as_bit(W := mpx_s1_3_state_reg_1);
mpx_s1_3_state_2_as_bit(W := mpx_s1_3_state_reg_2);
IF (mpx_s1_3_state_1_as_bit.B11 = FALSE) THEN
	mpx_s1_3_bypass_line_state := 'bypass_line1_off';
	mpx_s1_3_bypass_arrow_state := 'bypass_arrow_off';
	ELSE
		mpx_s1_3_bypass_line_state := 'bypass_line_on';
		mpx_s1_3_bypass_arrow_state := 'bypass_arrow_on';	
END_IF
IF (mpx_s1_3_state_1_as_bit.B15 = FALSE) THEN
	mpx_s1_3_output_state := 'arrow_off';
	ELSE
		mpx_s1_3_output_state := 'arrow_on';	
END_IF
IF (mpx_s1_3_state_2_as_bit.B12 = FALSE) THEN
	mpx_s1_3_input_state := 'arrow_off';
	ELSE
		mpx_s1_3_input_state := 'arrow_on';	
END_IF
IF (mpx_s1_3_state_1_as_bit.B13 = FALSE) THEN
	mpx_s1_3_battery_line_state := 'battery_line_off';
	mpx_s1_3_battery_arrow_state := 'battery_arrow_off';
	ELSE
		mpx_s1_3_battery_line_state := 'battery_line_on';
		mpx_s1_3_battery_arrow_state := 'battery_arrow_on';	
END_IF
IF ( (mpx_s1_3_state_2_as_bit.B13 = TRUE) OR (mpx_s1_3_state_2_as_bit.B14 = TRUE) OR (mpx_s1_3_state_2_as_bit.B15 = TRUE) ) THEN
	mpx_s1_3_alarm := TRUE;
	ELSE
		mpx_s1_3_alarm := FALSE;
END_IF

//Конвертация параметров MPX_s1_4
mpx_s1_4_in_freq_real               := mpx_s1_4_in_freq * 0.1;
mpx_s1_4_bypass_freq_real           := mpx_s1_4_bypass_freq * 0.1;
mpx_s1_4_output_i_1_real            := mpx_s1_4_output_i_1 * 0.1;
mpx_s1_4_output_i_2_real            := mpx_s1_4_output_i_2 * 0.1;
mpx_s1_4_output_i_3_real            := mpx_s1_4_output_i_3 * 0.1;
mpx_s1_4_output_active_power_1_real := mpx_s1_4_output_active_power_1 * 0.1;
mpx_s1_4_output_active_power_2_real := mpx_s1_4_output_active_power_2 * 0.1;
mpx_s1_4_output_active_power_3_real := mpx_s1_4_output_active_power_3 * 0.1;
mpx_s1_4_output_freq_real           := mpx_s1_4_output_freq * 0.1;
mpx_s1_4_battery_voltage_real       := mpx_s1_4_battery_voltage * 0.1;
mpx_s1_4_battery_current_real       := mpx_s1_4_battery_current * 0.1;

//Логика состояний MPX_s1_4
mpx_s1_4_state_1_as_bit(W := mpx_s1_4_state_reg_1);
mpx_s1_4_state_2_as_bit(W := mpx_s1_4_state_reg_2);
IF (mpx_s1_4_state_1_as_bit.B11 = FALSE) THEN
	mpx_s1_4_bypass_line_state := 'bypass_line1_off';
	mpx_s1_4_bypass_arrow_state := 'bypass_arrow_off';
	ELSE
		mpx_s1_4_bypass_line_state := 'bypass_line_on';
		mpx_s1_4_bypass_arrow_state := 'bypass_arrow_on';	
END_IF
IF (mpx_s1_4_state_1_as_bit.B15 = FALSE) THEN
	mpx_s1_4_output_state := 'arrow_off';
	ELSE
		mpx_s1_4_output_state := 'arrow_on';	
END_IF
IF (mpx_s1_4_state_2_as_bit.B12 = FALSE) THEN
	mpx_s1_4_input_state := 'arrow_off';
	ELSE
		mpx_s1_4_input_state := 'arrow_on';	
END_IF
IF (mpx_s1_4_state_1_as_bit.B13 = FALSE) THEN
	mpx_s1_4_battery_line_state := 'battery_line_off';
	mpx_s1_4_battery_arrow_state := 'battery_arrow_off';
	ELSE
		mpx_s1_4_battery_line_state := 'battery_line_on';
		mpx_s1_4_battery_arrow_state := 'battery_arrow_on';	
END_IF
IF ( (mpx_s1_4_state_2_as_bit.B13 = TRUE) OR (mpx_s1_4_state_2_as_bit.B14 = TRUE) OR (mpx_s1_4_state_2_as_bit.B15 = TRUE) ) THEN
	mpx_s1_4_alarm := TRUE;
	ELSE
		mpx_s1_4_alarm := FALSE;
END_IF

mpx_s1_all_power := mpx_s1_1_output_active_power_1_real + mpx_s1_1_output_active_power_2_real + mpx_s1_1_output_active_power_3_real + 
	                mpx_s1_2_output_active_power_1_real + mpx_s1_2_output_active_power_2_real + mpx_s1_2_output_active_power_3_real + 
                    mpx_s1_3_output_active_power_1_real + mpx_s1_3_output_active_power_2_real + mpx_s1_3_output_active_power_3_real + 
                    mpx_s1_4_output_active_power_1_real + mpx_s1_4_output_active_power_2_real + mpx_s1_4_output_active_power_3_real;
//------------------------------------MPX_S2-------------------------------------
//Конвертация параметров MPX_s2_1
mpx_s2_1_in_freq_real               := mpx_s2_1_in_freq * 0.1;
mpx_s2_1_bypass_freq_real           := mpx_s2_1_bypass_freq * 0.1;
mpx_s2_1_output_i_1_real            := mpx_s2_1_output_i_1 * 0.1;
mpx_s2_1_output_i_2_real            := mpx_s2_1_output_i_2 * 0.1;
mpx_s2_1_output_i_3_real            := mpx_s2_1_output_i_3 * 0.1;
mpx_s2_1_output_active_power_1_real := mpx_s2_1_output_active_power_1 * 0.1;
mpx_s2_1_output_active_power_2_real := mpx_s2_1_output_active_power_2 * 0.1;
mpx_s2_1_output_active_power_3_real := mpx_s2_1_output_active_power_3 * 0.1;
mpx_s2_1_output_freq_real           := mpx_s2_1_output_freq * 0.1;
mpx_s2_1_battery_voltage_real       := mpx_s2_1_battery_voltage * 0.1;
mpx_s2_1_battery_current_real       := mpx_s2_1_battery_current * 0.1;

//Логика состояний MPX_s2_1
mpx_s2_1_state_1_as_bit(W := mpx_s2_1_state_reg_1);
mpx_s2_1_state_2_as_bit(W := mpx_s2_1_state_reg_2);

IF (mpx_s2_1_state_1_as_bit.B15 = FALSE) THEN
	mpx_s2_1_output_state := 'arrow_off';
	ELSE
		mpx_s2_1_output_state := 'arrow_on';
		mpx_s2_state_string := "От всети";	
END_IF
IF (mpx_s2_1_state_2_as_bit.B12 = FALSE) THEN
	mpx_s2_1_input_state := 'arrow_off';
	ELSE
		mpx_s2_1_input_state := 'arrow_on';	
		mpx_s2_state_string := "От сети";
END_IF
IF (mpx_s2_1_state_1_as_bit.B13 = FALSE) THEN
	mpx_s2_1_battery_line_state := 'battery_line_off';
	mpx_s2_1_battery_arrow_state := 'battery_arrow_off';
	ELSE
		mpx_s2_1_battery_line_state := 'battery_line_on';
		mpx_s2_1_battery_arrow_state := 'battery_arrow_on';	
		mpx_s2_state_string := "От АКБ";
END_IF
IF (mpx_s2_1_state_1_as_bit.B11 = FALSE) THEN
	mpx_s2_1_bypass_line_state := 'bypass_line1_off';
	mpx_s2_1_bypass_arrow_state := 'bypass_arrow_off';
	ELSE
		mpx_s2_1_bypass_line_state := 'bypass_line_on';
		mpx_s2_1_bypass_arrow_state := 'bypass_arrow_on';
		mpx_s2_state_string := "Байпас";	
END_IF
IF ( (mpx_s2_1_state_2_as_bit.B13 = TRUE) OR (mpx_s2_1_state_2_as_bit.B14 = TRUE) OR (mpx_s2_1_state_2_as_bit.B15 = TRUE) ) THEN
	mpx_s2_1_alarm := TRUE;
	ELSE
		mpx_s2_1_alarm := FALSE;
END_IF

//Конвертация параметров MPX_s2_2
mpx_s2_2_in_freq_real               := mpx_s2_2_in_freq * 0.1;
mpx_s2_2_bypass_freq_real           := mpx_s2_2_bypass_freq * 0.1;
mpx_s2_2_output_i_1_real            := mpx_s2_2_output_i_1 * 0.1;
mpx_s2_2_output_i_2_real            := mpx_s2_2_output_i_2 * 0.1;
mpx_s2_2_output_i_3_real            := mpx_s2_2_output_i_3 * 0.1;
mpx_s2_2_output_active_power_1_real := mpx_s2_2_output_active_power_1 * 0.1;
mpx_s2_2_output_active_power_2_real := mpx_s2_2_output_active_power_2 * 0.1;
mpx_s2_2_output_active_power_3_real := mpx_s2_2_output_active_power_3 * 0.1;
mpx_s2_2_output_freq_real           := mpx_s2_2_output_freq * 0.1;
mpx_s2_2_battery_voltage_real       := mpx_s2_2_battery_voltage * 0.1;
mpx_s2_2_battery_current_real       := mpx_s2_2_battery_current * 0.1;

//Логика состояний MPX_S2_2
mpx_s2_2_state_1_as_bit(W := mpx_s2_2_state_reg_1);
mpx_s2_2_state_2_as_bit(W := mpx_s2_2_state_reg_2);
IF (mpx_s2_2_state_1_as_bit.B11 = FALSE) THEN
	mpx_s2_2_bypass_line_state := 'bypass_line1_off';
	mpx_s2_2_bypass_arrow_state := 'bypass_arrow_off';
	ELSE
		mpx_s2_2_bypass_line_state := 'bypass_line_on';
		mpx_s2_2_bypass_arrow_state := 'bypass_arrow_on';	
END_IF
IF (mpx_s2_2_state_1_as_bit.B15 = FALSE) THEN
	mpx_s2_2_output_state := 'arrow_off';
	ELSE
		mpx_s2_2_output_state := 'arrow_on';	
END_IF
IF (mpx_s2_2_state_2_as_bit.B12 = FALSE) THEN
	mpx_s2_2_input_state := 'arrow_off';
	ELSE
		mpx_s2_2_input_state := 'arrow_on';	
END_IF
IF (mpx_s2_2_state_1_as_bit.B13 = FALSE) THEN
	mpx_s2_2_battery_line_state := 'battery_line_off';
	mpx_s2_2_battery_arrow_state := 'battery_arrow_off';
	ELSE
		mpx_s2_2_battery_line_state := 'battery_line_on';
		mpx_s2_2_battery_arrow_state := 'battery_arrow_on';	
END_IF
IF ( (mpx_s2_2_state_2_as_bit.B13 = TRUE) OR (mpx_s2_2_state_2_as_bit.B14 = TRUE) OR (mpx_s2_2_state_2_as_bit.B15 = TRUE) ) THEN
	mpx_s2_2_alarm := TRUE;
	ELSE
		mpx_s2_2_alarm := FALSE;
END_IF

//Конвертация параметров MPX_s2_3
mpx_s2_3_in_freq_real               := mpx_s2_3_in_freq * 0.1;
mpx_s2_3_bypass_freq_real           := mpx_s2_3_bypass_freq * 0.1;
mpx_s2_3_output_i_1_real            := mpx_s2_3_output_i_1 * 0.1;
mpx_s2_3_output_i_2_real            := mpx_s2_3_output_i_2 * 0.1;
mpx_s2_3_output_i_3_real            := mpx_s2_3_output_i_3 * 0.1;
mpx_s2_3_output_active_power_1_real := mpx_s2_3_output_active_power_1 * 0.1;
mpx_s2_3_output_active_power_2_real := mpx_s2_3_output_active_power_2 * 0.1;
mpx_s2_3_output_active_power_3_real := mpx_s2_3_output_active_power_3 * 0.1;
mpx_s2_3_output_freq_real           := mpx_s2_3_output_freq * 0.1;
mpx_s2_3_battery_voltage_real       := mpx_s2_3_battery_voltage * 0.1;
mpx_s2_3_battery_current_real       := mpx_s2_3_battery_current * 0.1;

//Логика состояний MPX_S2_3
mpx_s2_3_state_1_as_bit(W := mpx_s2_3_state_reg_1);
mpx_s2_3_state_2_as_bit(W := mpx_s2_3_state_reg_2);
IF (mpx_s2_3_state_1_as_bit.B11 = FALSE) THEN
	mpx_s2_3_bypass_line_state := 'bypass_line1_off';
	mpx_s2_3_bypass_arrow_state := 'bypass_arrow_off';
	ELSE
		mpx_s2_3_bypass_line_state := 'bypass_line_on';
		mpx_s2_3_bypass_arrow_state := 'bypass_arrow_on';	
END_IF
IF (mpx_s2_3_state_1_as_bit.B15 = FALSE) THEN
	mpx_s2_3_output_state := 'arrow_off';
	ELSE
		mpx_s2_3_output_state := 'arrow_on';	
END_IF
IF (mpx_s2_3_state_2_as_bit.B12 = FALSE) THEN
	mpx_s2_3_input_state := 'arrow_off';
	ELSE
		mpx_s2_3_input_state := 'arrow_on';	
END_IF
IF (mpx_s2_3_state_1_as_bit.B13 = FALSE) THEN
	mpx_s2_3_battery_line_state := 'battery_line_off';
	mpx_s2_3_battery_arrow_state := 'battery_arrow_off';
	ELSE
		mpx_s2_3_battery_line_state := 'battery_line_on';
		mpx_s2_3_battery_arrow_state := 'battery_arrow_on';	
END_IF
IF ( (mpx_s2_3_state_2_as_bit.B13 = TRUE) OR (mpx_s2_3_state_2_as_bit.B14 = TRUE) OR (mpx_s2_3_state_2_as_bit.B15 = TRUE) ) THEN
	mpx_s2_3_alarm := TRUE;
	ELSE
		mpx_s2_3_alarm := FALSE;
END_IF

//Конвертация параметров MPX_s2_4
mpx_s2_4_in_freq_real               := mpx_s2_4_in_freq * 0.1;
mpx_s2_4_bypass_freq_real           := mpx_s2_4_bypass_freq * 0.1;
mpx_s2_4_output_i_1_real            := mpx_s2_4_output_i_1 * 0.1;
mpx_s2_4_output_i_2_real            := mpx_s2_4_output_i_2 * 0.1;
mpx_s2_4_output_i_3_real            := mpx_s2_4_output_i_3 * 0.1;
mpx_s2_4_output_active_power_1_real := mpx_s2_4_output_active_power_1 * 0.1;
mpx_s2_4_output_active_power_2_real := mpx_s2_4_output_active_power_2 * 0.1;
mpx_s2_4_output_active_power_3_real := mpx_s2_4_output_active_power_3 * 0.1;
mpx_s2_4_output_freq_real           := mpx_s2_4_output_freq * 0.1;
mpx_s2_4_battery_voltage_real       := mpx_s2_4_battery_voltage * 0.1;
mpx_s2_4_battery_current_real       := mpx_s2_4_battery_current * 0.1;

//Логика состояний MPX_S2_4
mpx_s2_4_state_1_as_bit(W := mpx_s2_4_state_reg_1);
mpx_s2_4_state_2_as_bit(W := mpx_s2_4_state_reg_2);
IF (mpx_s2_4_state_1_as_bit.B11 = FALSE) THEN
	mpx_s2_4_bypass_line_state := 'bypass_line1_off';
	mpx_s2_4_bypass_arrow_state := 'bypass_arrow_off';
	ELSE
		mpx_s2_4_bypass_line_state := 'bypass_line_on';
		mpx_s2_4_bypass_arrow_state := 'bypass_arrow_on';	
END_IF
IF (mpx_s2_4_state_1_as_bit.B15 = FALSE) THEN
	mpx_s2_4_output_state := 'arrow_off';
	ELSE
		mpx_s2_4_output_state := 'arrow_on';	
END_IF
IF (mpx_s2_4_state_2_as_bit.B12 = FALSE) THEN
	mpx_s2_4_input_state := 'arrow_off';
	ELSE
		mpx_s2_4_input_state := 'arrow_on';	
END_IF
IF (mpx_s2_4_state_1_as_bit.B13 = FALSE) THEN
	mpx_s2_4_battery_line_state := 'battery_line_off';
	mpx_s2_4_battery_arrow_state := 'battery_arrow_off';
	ELSE
		mpx_s2_4_battery_line_state := 'battery_line_on';
		mpx_s2_4_battery_arrow_state := 'battery_arrow_on';	
END_IF
IF ( (mpx_s2_4_state_2_as_bit.B13 = TRUE) OR (mpx_s2_4_state_2_as_bit.B14 = TRUE) OR (mpx_s2_4_state_2_as_bit.B15 = TRUE) ) THEN
	mpx_s2_4_alarm := TRUE;
	ELSE
		mpx_s2_4_alarm := FALSE;
END_IF

mpx_s2_all_power := mpx_s2_1_output_active_power_1_real + mpx_s2_1_output_active_power_2_real + mpx_s2_1_output_active_power_3_real + 
	                mpx_s2_2_output_active_power_1_real + mpx_s2_2_output_active_power_2_real + mpx_s2_2_output_active_power_3_real + 
                    mpx_s2_3_output_active_power_1_real + mpx_s2_3_output_active_power_2_real + mpx_s2_3_output_active_power_3_real + 
                    mpx_s2_4_output_active_power_1_real + mpx_s2_4_output_active_power_2_real + mpx_s2_4_output_active_power_3_real;

END_PROGRAM

// CODESYS_Control_for_Raspberry_Pi/Application/GPIO_HANDLER
PROGRAM GPIO_HANDLER
VAR
	
	IN_1: BOOL; // Нарушение ШОС
	
	IN_2: BOOL; // Пожар
	
	IN_3: BOOL; // Неисправность ШОС
	
	IN_4: BOOL; // Наличие напряжения на 1 вводе
	
	IN_5: BOOL; // Наличие напряжения на 2 вводе
	
	IN_6: BOOL; // QS1 в первом положении
	
	IN_7: BOOL; // QS1 во втором положении
	
	IN_8: BOOL; // QS2 в первом положении
	
	IN_9: BOOL; // QS2 во втором положении
	
	IN_10: BOOL; // QS3 в первом положении
	
	IN_11: BOOL; // QS3 во втором положении
	IN_12: BOOL;
END_VAR

IN_1 := NOT(IN_1);
IN_2 := NOT(IN_2);
IN_3 := NOT(IN_3);
IN_4 := NOT(IN_4);
IN_5 := NOT(IN_5);
IN_6 := NOT(IN_6);
IN_7 := NOT(IN_7);
IN_8 := NOT(IN_8);
IN_9 := NOT(IN_9);
IN_10 := NOT(IN_10);
IN_11 := NOT(IN_11);
IN_12 := NOT(IN_12);

END_PROGRAM

// CODESYS_Control_for_Raspberry_Pi/Application/AlarmChecker
PROGRAM AlarmChecker
VAR
	MIN_VOLTAGE : WORD := 50;
	
	ups_s1_in_v_alarm : BOOL;
	ups_s2_in_v_alarm : BOOL;
	ups_a1_in_v_alarm : BOOL;
	ups_a2_in_v_alarm : BOOL;
	
	ups_s1_out_v_alarm : BOOL;
	ups_s2_out_v_alarm : BOOL;
	ups_a1_out_v_alarm : BOOL;
	ups_a2_out_v_alarm : BOOL;
	
	shasn_alarm        : BOOL;
	schrpa_alarm       : BOOL;
	schrps_alarm       : BOOL;
END_VAR

//Авария входного напряжения ИБПС1
IF( (PLC_PRG.mpx_s1_1_in_v_1 < MIN_VOLTAGE) OR (PLC_PRG.mpx_s1_1_in_v_2 < MIN_VOLTAGE) OR (PLC_PRG.mpx_s1_1_in_v_3 < MIN_VOLTAGE)
OR  (PLC_PRG.mpx_s1_2_in_v_1 < MIN_VOLTAGE) OR (PLC_PRG.mpx_s1_2_in_v_2 < MIN_VOLTAGE) OR (PLC_PRG.mpx_s1_2_in_v_3 < MIN_VOLTAGE)
OR  (PLC_PRG.mpx_s1_3_in_v_1 < MIN_VOLTAGE) OR (PLC_PRG.mpx_s1_3_in_v_2 < MIN_VOLTAGE) OR (PLC_PRG.mpx_s1_3_in_v_3 < MIN_VOLTAGE)
OR  (PLC_PRG.mpx_s1_4_in_v_1 < MIN_VOLTAGE) OR (PLC_PRG.mpx_s1_4_in_v_2 < MIN_VOLTAGE) OR (PLC_PRG.mpx_s1_4_in_v_3 < MIN_VOLTAGE) ) THEN
	ups_s1_in_v_alarm := TRUE;
	ELSE
		ups_s1_in_v_alarm := FALSE;
END_IF

//Авария входного напряжения ИБПС2
IF( (PLC_PRG.mpx_s2_1_in_v_1 < MIN_VOLTAGE) OR (PLC_PRG.mpx_s2_1_in_v_2 < MIN_VOLTAGE) OR (PLC_PRG.mpx_s2_1_in_v_3 < MIN_VOLTAGE)
OR  (PLC_PRG.mpx_s2_2_in_v_1 < MIN_VOLTAGE) OR (PLC_PRG.mpx_s2_2_in_v_2 < MIN_VOLTAGE) OR (PLC_PRG.mpx_s2_2_in_v_3 < MIN_VOLTAGE)
OR  (PLC_PRG.mpx_s2_3_in_v_1 < MIN_VOLTAGE) OR (PLC_PRG.mpx_s2_3_in_v_2 < MIN_VOLTAGE) OR (PLC_PRG.mpx_s2_3_in_v_3 < MIN_VOLTAGE)
OR  (PLC_PRG.mpx_s2_4_in_v_1 < MIN_VOLTAGE) OR (PLC_PRG.mpx_s2_4_in_v_2 < MIN_VOLTAGE) OR (PLC_PRG.mpx_s2_4_in_v_3 < MIN_VOLTAGE) ) THEN
	ups_s2_in_v_alarm := TRUE;
	ELSE
		ups_s2_in_v_alarm := FALSE;
END_IF

//Авария входного напряжения ИБПА1
IF( (PLC_PRG.mpx_a1_1_in_v_1 < MIN_VOLTAGE) OR (PLC_PRG.mpx_a1_1_in_v_2 < MIN_VOLTAGE) OR (PLC_PRG.mpx_a1_1_in_v_3 < MIN_VOLTAGE)
OR  (PLC_PRG.mpx_a1_2_in_v_1 < MIN_VOLTAGE) OR (PLC_PRG.mpx_a1_2_in_v_2 < MIN_VOLTAGE) OR (PLC_PRG.mpx_a1_2_in_v_3 < MIN_VOLTAGE) ) THEN
	ups_a1_in_v_alarm := TRUE;
	ELSE
		ups_a1_in_v_alarm := FALSE;
END_IF

//Авария входного напряжения ИБПА2
IF( (PLC_PRG.mpx_a2_1_in_v_1 < MIN_VOLTAGE) OR (PLC_PRG.mpx_a2_1_in_v_2 < MIN_VOLTAGE) OR (PLC_PRG.mpx_a2_1_in_v_3 < MIN_VOLTAGE)
OR  (PLC_PRG.mpx_a2_2_in_v_1 < MIN_VOLTAGE) OR (PLC_PRG.mpx_a2_2_in_v_2 < MIN_VOLTAGE) OR (PLC_PRG.mpx_a2_2_in_v_3 < MIN_VOLTAGE) ) THEN
	ups_a2_in_v_alarm := TRUE;
	ELSE
		ups_a2_in_v_alarm := FALSE;
END_IF

//------------------------------------------------------------------------------

//Авария выходного напряжения ИБПС1
IF( (PLC_PRG.mpx_s1_1_output_v_1 < MIN_VOLTAGE) OR (PLC_PRG.mpx_s1_1_output_v_2 < MIN_VOLTAGE) OR (PLC_PRG.mpx_s1_1_output_v_3 < MIN_VOLTAGE)
OR  (PLC_PRG.mpx_s1_2_output_v_1 < MIN_VOLTAGE) OR (PLC_PRG.mpx_s1_2_output_v_2 < MIN_VOLTAGE) OR (PLC_PRG.mpx_s1_2_output_v_3 < MIN_VOLTAGE)
OR  (PLC_PRG.mpx_s1_3_output_v_1 < MIN_VOLTAGE) OR (PLC_PRG.mpx_s1_3_output_v_2 < MIN_VOLTAGE) OR (PLC_PRG.mpx_s1_3_output_v_3 < MIN_VOLTAGE)
OR  (PLC_PRG.mpx_s1_4_output_v_1 < MIN_VOLTAGE) OR (PLC_PRG.mpx_s1_4_output_v_2 < MIN_VOLTAGE) OR (PLC_PRG.mpx_s1_4_output_v_3 < MIN_VOLTAGE) ) THEN
	ups_s1_out_v_alarm := TRUE;
	ELSE
		ups_s1_out_v_alarm := FALSE;
END_IF

//Авария выходного напряжения ИБПС2
IF( (PLC_PRG.mpx_s2_1_output_v_1 < MIN_VOLTAGE) OR (PLC_PRG.mpx_s2_1_output_v_2 < MIN_VOLTAGE) OR (PLC_PRG.mpx_s2_1_output_v_3 < MIN_VOLTAGE)
OR  (PLC_PRG.mpx_s2_2_output_v_1 < MIN_VOLTAGE) OR (PLC_PRG.mpx_s2_2_output_v_2 < MIN_VOLTAGE) OR (PLC_PRG.mpx_s2_2_output_v_3 < MIN_VOLTAGE)
OR  (PLC_PRG.mpx_s2_3_output_v_1 < MIN_VOLTAGE) OR (PLC_PRG.mpx_s2_3_output_v_2 < MIN_VOLTAGE) OR (PLC_PRG.mpx_s2_3_output_v_3 < MIN_VOLTAGE)
OR  (PLC_PRG.mpx_s2_4_output_v_1 < MIN_VOLTAGE) OR (PLC_PRG.mpx_s2_4_output_v_2 < MIN_VOLTAGE) OR (PLC_PRG.mpx_s2_4_output_v_3 < MIN_VOLTAGE) ) THEN
	ups_s2_out_v_alarm := TRUE;
	ELSE
		ups_s2_out_v_alarm := FALSE;
END_IF

//Авария выходного напряжения ИБПА1
IF( (PLC_PRG.mpx_a1_1_output_v_1 < MIN_VOLTAGE)
OR  (PLC_PRG.mpx_a1_2_output_v_1 < MIN_VOLTAGE) ) THEN
	ups_a1_out_v_alarm := TRUE;
	ELSE
		ups_a1_out_v_alarm := FALSE;
END_IF

//Авария выходного напряжения ИБПА2
IF( (PLC_PRG.mpx_a2_1_output_v_1 < MIN_VOLTAGE)
OR  (PLC_PRG.mpx_a2_2_output_v_1 < MIN_VOLTAGE) ) THEN
	ups_a2_out_v_alarm := TRUE;
	ELSE
		ups_a2_out_v_alarm := FALSE;
END_IF

//Авария ШАСН
IF ( (PLC_PRG.mv110_in_0_in_main_present = FALSE) OR (PLC_PRG.mv110_in_1_in_reserve_present = FALSE) ) THEN
	shasn_alarm := TRUE;
	ELSE
		shasn_alarm := FALSE;
END_IF

//Авария ЩРПА
IF ( (GPIO_HANDLER.IN_4 = FALSE) OR (GPIO_HANDLER.IN_5 = FALSE) ) THEN
	schrpa_alarm := TRUE;
	ELSE
		schrpa_alarm := FALSE;
END_IF

//Авария ЩРПС
IF ( (PLC_PRG.mv110_in_7_gp1_u_fault = TRUE) OR (PLC_PRG.mv110_in_8_gp2_u_fault = TRUE) ) THEN
	schrps_alarm := TRUE;
	ELSE
		schrps_alarm := FALSE;
END_IF

END_PROGRAM

// CODESYS_Control_for_Raspberry_Pi/Application/BusReinit
PROGRAM BusReinit
VAR
	BL1 : BLINK;
	BL2 : BLINK;
END_VAR



IF MV_110.xError THEN 
	BL1(enable:=TRUE, timelow:=T#500MS, timehigh:=T#1000MS);
	MV_110.xReset:=BL1.OUT; 
	ModbusMaster.xResetComPort := TRUE;
ELSE 
	BL1(enable:=FALSE, timelow:=T#500MS, timehigh:=T#1000MS);
	MV_110.xReset:= FALSE;
	ModbusMaster.xResetComPort := FALSE; 
END_IF;

IF PLC.xError THEN 
	BL2(enable:=TRUE, timelow:=T#500MS, timehigh:=T#1000MS);
	PLC.xReset:=BL2.OUT; 
	ModbusMaster.xResetComPort := TRUE;
ELSE 
	BL2(enable:=FALSE, timelow:=T#500MS, timehigh:=T#1000MS);
	PLC.xReset:= FALSE;
	ModbusMaster.xResetComPort := FALSE; 
END_IF;

END_PROGRAM

// CODESYS_Control_for_Raspberry_Pi/Application/InterviewState
PROGRAM InterviewState
VAR
	//Переменные состояния опроса модулей ИБПС 1
	MPX_S1_1_State : BOOL;
	MPX_S1_2_State : BOOL;
	MPX_S1_3_State : BOOL;
	MPX_S1_4_State : BOOL;
	MPX_S1_State   : BOOL;	

	//Переменные состояния опроса модулей ИБПС 2
	MPX_s2_1_State : BOOL;
	MPX_S2_2_State : BOOL;
	MPX_S2_3_State : BOOL;
	MPX_S2_4_State : BOOL;
	MPX_S2_State   : BOOL;
	
	//Переменные состояния опроса модулей ИБПА 1
	MPX_A1_1_State : BOOL;
	MPX_A1_2_State : BOOL;
	MPX_A1_3_State : BOOL;
	MPX_A1_4_State : BOOL;
	MPX_A1_State   : BOOL;
	
	//Переменные состояния опроса модулей ИБПА 2
	MPX_A2_1_State : BOOL;
	MPX_A2_2_State : BOOL;
	MPX_A2_3_State : BOOL;
	MPX_A2_4_State : BOOL;
	MPX_A2_State   : BOOL;
		
END_VAR

MPX_s2_1_State := MPX_s2_1.xError;
MPX_S2_2_State := MPX_S2_2.xError;
MPX_S2_3_State := MPX_S2_3.xError;
MPX_S2_4_State := MPX_S2_4.xError;

IF ( (MPX_s2_1_State = TRUE) OR (MPX_S2_2_State = TRUE) OR (MPX_S2_3_State = TRUE) OR (MPX_S2_4_State = TRUE) ) THEN
	MPX_S2_State := TRUE;
ELSE
	MPX_S2_State := FALSE;	
END_IF

MPX_s1_1_State := MPX_s1_1.xError;
MPX_s1_2_State := MPX_s1_2.xError;
MPX_s1_3_State := MPX_s1_3.xError;
MPX_s1_4_State := MPX_s1_4.xError;

IF ( (MPX_s1_1_State = TRUE) OR (MPX_s1_2_State = TRUE) OR (MPX_s1_3_State = TRUE) OR (MPX_s1_4_State = TRUE) ) THEN
	MPX_s1_State := TRUE;
ELSE
	MPX_s1_State := FALSE;	
END_IF

END_PROGRAM

// CODESYS_Control_for_Raspberry_Pi/Application/visualization/monitoring
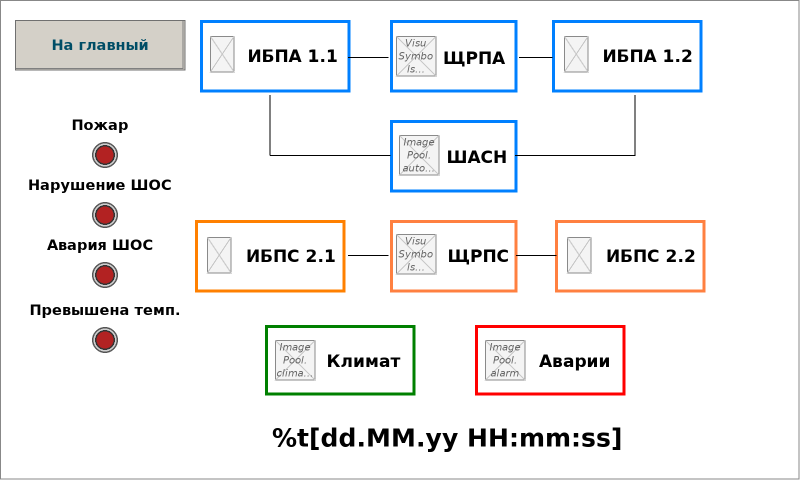
VISUALIZATION monitoring  // 800x480, background image ImagePool.bg_800
    Lamp1 (90,140 30x30), variable: GPIO_HANDLER.IN_2, style: Lamp-Lamp1-Red
    Rectangle (20,110 160x30), "Пожар"
    Lamp1 (90,200 30x30), variable: GPIO_HANDLER.IN_1, style: Lamp-Lamp1-Red
    Rectangle (20,170 160x30), "Нарушение ШОС"
    Lamp1 (90,260 30x30), variable: GPIO_HANDLER.IN_3, style: Lamp-Lamp1-Red
    Rectangle (20,230 160x30), "Авария ШОС"
    Lamp1 (90,325 30x30), variable: PLC_PRG.climate_temp_excess, style: Lamp-Lamp1-Red
    Rectangle (20,295 170x30), "Превышена темп."
    Group (390,220 127x72)
        OnMouseClick:  Assign=schrps, Type=Assignment
        RoundedRectangle (0,0 127x72), colour toggle: AlarmChecker.schrps_alarm
        RoundedRectangle (51,20 75x32), "ЩРПС"
            OnMouseClick:  Assign=ups_s2, Type=Assignment
        Image (6,14 40x40), image: VisuSymbols.Symbols.TreeDown
    Group (390,20 127x72)
        OnMouseClick:  Assign=schrpa, Type=Assignment
        RoundedRectangle (0,0 127x72), colour toggle: AlarmChecker.schrpa_alarm
            OnMouseClick:  Assign=ups_s2, Type=Assignment
        Image (6,16 40x40), image: VisuSymbols.Symbols.TreeDown
        RoundedRectangle (51,22 66x32), "ЩРПА"
            OnMouseClick:  Assign=ups_s2, Type=Assignment
    Group (390,120 127x72)
        OnMouseClick:  Assign=shasn, Type=Assignment
        RoundedRectangle (0,0 127x72), colour toggle: AlarmChecker.shasn_alarm
            OnMouseClick:  Assign=ups_s2, Type=Assignment
        RoundedRectangle (48,21 78x32), "ШАСН"
            OnMouseClick:  Assign=ups_s2, Type=Assignment
        Image (9,15 40x40), image: ImagePool.automation-512
    Button (15,20 170x50), "На главный"
        OnMouseClick:  Assign=main, Type=Assignment
    Group (265,325 150x70)
        OnMouseClick:  Assign=climate, Type=Assignment
        RoundedRectangle (0,0 150x70)
        RoundedRectangle (55,20 87x32), "Климат"
            OnMouseClick:  Assign=ups_s2, Type=Assignment
        Image (10,15 40x40), image: ImagePool.climate
    Group (475,325 150x70)
        OnMouseClick:  Assign=alarm, Type=Assignment
        RoundedRectangle (0,0 150x70)
        RoundedRectangle (55,20 90x32), "Аварии"
            OnMouseClick:  Assign=ups_s2, Type=Assignment
        Image (10,15 40x40), image: ImagePool.alarm
    Group (195,220 150x72)
        OnMouseClick:  Assign=ups_s1, Type=Assignment
        RoundedRectangle (0,0 150x72), colour toggle: AlarmChecker.ups_s1_in_v_alarm
            OnMouseClick:  Assign=ups_s2, Type=Assignment
        RoundedRectangle (45,20 102x32), "ИБПС 2.1"
            OnMouseClick:  Assign=ups_s2, Type=Assignment
        Image (12,17 24x36), image: ImagePool.mini_ups
    Group (555,220 150x72)
        OnMouseClick:  Assign=ups_s2, Type=Assignment
        RoundedRectangle (0,0 150x72), colour toggle: AlarmChecker.ups_s2_in_v_alarm
            OnMouseClick:  Assign=ups_s2, Type=Assignment
        RoundedRectangle (45,20 102x32), "ИБПС 2.2"
            OnMouseClick:  Assign=ups_s2, Type=Assignment
        Image (12,17 24x36), image: ImagePool.mini_ups
    Group (200,20 150x72)
        OnMouseClick:  Assign=ups_a1, Type=Assignment
        RoundedRectangle (0,0 150x72), colour toggle: AlarmChecker.ups_a1_in_v_alarm
            OnMouseClick:  Assign=ups_s2, Type=Assignment
        RoundedRectangle (42,20 102x32), "ИБПА 1.1"
            OnMouseClick:  Assign=ups_s2, Type=Assignment
        Image (10,16 24x36), image: ImagePool.mini_ups
    Rectangle (260,415 375x45), "%t[dd.MM.yy HH:mm:ss]"
    Group (552,20 150x72)
        OnMouseClick:  Assign=ups_a2, Type=Assignment
        RoundedRectangle (0,0 150x72), colour toggle: AlarmChecker.ups_a2_in_v_alarm
            OnMouseClick:  Assign=ups_s2, Type=Assignment
        RoundedRectangle (45,20 102x32), "ИБПА 1.2"
            OnMouseClick:  Assign=ups_s2, Type=Assignment
        Image (12,16 24x36), image: ImagePool.mini_ups
    Line (640,130)
    Line (635,155) (635,95)
    Line (515,155) (635,155)
    Line (270,155) (390,155)
    Line (270,155) (270,95)
    Line (348,57) (388,57)
    Line (519,57) (552,57)
    Line (348,255) (388,255)
    Line (516,255) (556,255)
    hotkey  Id=481037385728, Key=KeyDown=True, KeyName=0, VisuElemId=148
    hotkey  Id=481038434304, Key=KeyName=0, VisuElemId=148
END_VISUALIZATION

// CODESYS_Control_for_Raspberry_Pi/Application/visualization/ups_s2/ups_s2_m1_state
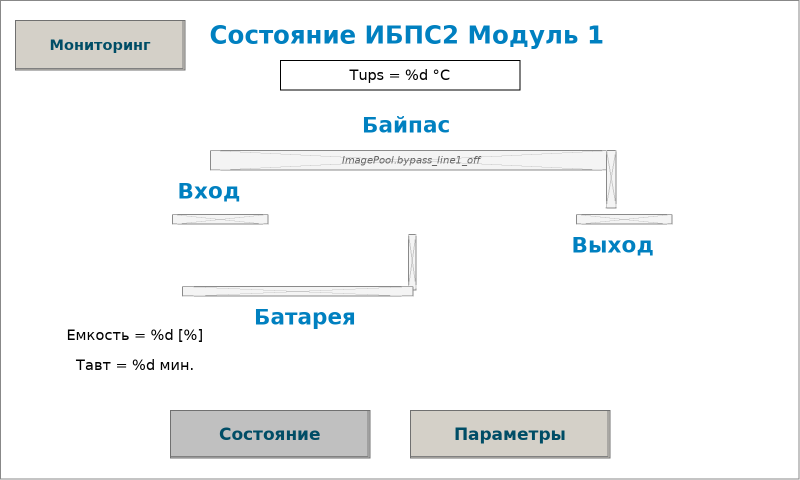
VISUALIZATION ups_s2_m1_state  // 800x480, background image ImagePool.mpx_state_bg
    Rectangle (204,20 406x30), "Состояние ИБПС2 Модуль 1"
    Button (410,410 200x48), "Параметры"
        OnMouseClick:  Assign=ups_s2_m1_params, Type=Assignment
    Button (170,410 200x48), "Состояние", pressed state: PLC_PRG.var_true
    Rectangle (350,110 112x30), "Байпас"
    Rectangle (246,302 118x30), "Батарея"
    Rectangle (166,176 86x30), "Вход"
    Rectangle (560,230 106x30), "Выход"
    Rectangle (280,60 240x30), "Tups = %d °С", text variable: PLC_PRG.mpx_s2_1_temp
    Rectangle (30,320 210x30), "Емкость = %d [%]", text variable: PLC_PRG.mpx_s2_1_battery_capacity
    Rectangle (30,350 210x30), "Tавт = %d мин.", text variable: PLC_PRG.mpx_s2_1_battery_time
    Image (210,150 402x20), image: ImagePool.bypass_line1_off
        p84334746: PLC_PRG.mpx_s2_1_bypass_line_state
    Image (606,150 10x58), image: ImagePool.bypass_arrow_off
        p84334746: PLC_PRG.mpx_s2_1_bypass_arrow_state
    Image (576,214 96x10), image: ImagePool.arrow_off
        p84334746: PLC_PRG.mpx_s2_1_output_state
    Image (172,214 96x10), image: ImagePool.arrow_off
        p84334746: PLC_PRG.mpx_s2_1_input_state
    Image (408,234 8x56), image: ImagePool.battery_arrow_off
        p84334746: PLC_PRG.mpx_s2_1_battery_arrow_state
    Image (182,286 231x10), image: ImagePool.battery_line_off
        p84334746: PLC_PRG.mpx_s2_1_battery_line_state
    Button (15,20 170x50), "Мониторинг"
        OnMouseClick:  Assign=monitoring, Type=Assignment
    hotkey  Id=481037385728, Key=KeyDown=True, KeyName=0, VisuElemId=38
    hotkey  Id=481038434304, Key=KeyName=0, VisuElemId=38
END_VISUALIZATION

// CODESYS_Control_for_Raspberry_Pi/Application/visualization/ups_s2/ups_s2_m1_params
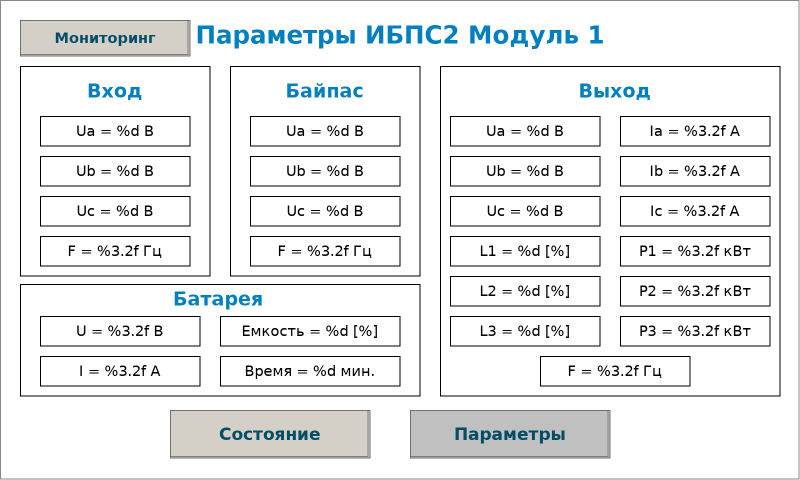
VISUALIZATION ups_s2_m1_params  // 800x480, background image ImagePool.bg_800
    Rectangle (186,20 428x30), "Параметры ИБПC2 Модуль 1"
    Button (170,410 200x48), "Состояние"
        OnMouseClick:  Assign=ups_s2_m1_state, Type=Assignment
    Button (410,410 200x48), "Параметры", pressed state: PLC_PRG.var_true
    Button (20,20 170x36), "Мониторинг"
        OnMouseClick:  Assign=monitoring, Type=Assignment
    Rectangle (20,66 190x210)
    Rectangle (440,66 340x330)
    Rectangle (30,76 170x30), "Вход"
    Rectangle (40,116 150x30), "Ua = %d В", text variable: PLC_PRG.mpx_s2_1_in_v_1
    Rectangle (40,156 150x30), "Ub = %d В", text variable: PLC_PRG.mpx_s2_1_in_v_2
    Rectangle (40,196 150x30), "Uc = %d В", text variable: PLC_PRG.mpx_s2_1_in_v_3
    Rectangle (40,236 150x30), "F = %3.2f Гц", text variable: PLC_PRG.mpx_s2_1_in_freq_real
    Rectangle (230,66 190x210)
    Rectangle (240,76 170x30), "Байпас"
    Rectangle (250,116 150x30), "Ua = %d В", text variable: PLC_PRG.mpx_s2_1_bypass_v_1
    Rectangle (250,156 150x30), "Ub = %d В", text variable: PLC_PRG.mpx_s2_1_bypass_v_2
    Rectangle (250,196 150x30), "Uc = %d В", text variable: PLC_PRG.mpx_s2_1_bypass_v_3
    Rectangle (250,236 150x30), "F = %3.2f Гц", text variable: PLC_PRG.mpx_s2_1_bypass_freq_real
    Rectangle (460,76 310x30), "Выход"
    Rectangle (450,116 150x30), "Ua = %d В", text variable: PLC_PRG.mpx_s2_1_output_v_1
    Rectangle (450,156 150x30), "Ub = %d В", text variable: PLC_PRG.mpx_s2_1_output_v_2
    Rectangle (450,196 150x30), "Uc = %d В", text variable: PLC_PRG.mpx_s2_1_output_v_3
    Rectangle (620,116 150x30), "Ia = %3.2f A", text variable: PLC_PRG.mpx_s2_1_output_i_1_real
    Rectangle (620,156 150x30), "Ib = %3.2f A", text variable: PLC_PRG.mpx_s2_1_output_i_2_real
    Rectangle (620,196 150x30), "Ic = %3.2f A", text variable: PLC_PRG.mpx_s2_1_output_i_3_real
    Rectangle (450,236 150x30), "L1 = %d [%]", text variable: PLC_PRG.mpx_s2_1_load_ph_1
    Rectangle (450,276 150x30), "L2 = %d [%]", text variable: PLC_PRG.mpx_s2_1_load_ph_2
    Rectangle (450,316 150x30), "L3 = %d [%]", text variable: PLC_PRG.mpx_s2_1_load_ph_3
    Rectangle (620,236 150x30), "P1 = %3.2f кВт", text variable: PLC_PRG.mpx_s2_1_output_active_power_1_real
    Rectangle (620,276 150x30), "P2 = %3.2f кВт", text variable: PLC_PRG.mpx_s2_1_output_active_power_2_real
    Rectangle (620,316 150x30), "P3 = %3.2f кВт", text variable: PLC_PRG.mpx_s2_1_output_active_power_3_real
    Rectangle (540,356 150x30), "F = %3.2f Гц", text variable: PLC_PRG.mpx_s2_1_output_freq_real
    Rectangle (20,284 400x112)
    Rectangle (30,290 376x18), "Батарея"
    Rectangle (40,316 160x30), "U = %3.2f В", text variable: PLC_PRG.mpx_s2_1_battery_voltage_real
    Rectangle (40,356 160x30), "I = %3.2f A", text variable: PLC_PRG.mpx_s2_1_battery_current_real
    Rectangle (220,316 180x30), "Емкость = %d [%]", text variable: PLC_PRG.mpx_s2_1_battery_capacity
    Rectangle (220,356 180x30), "Время = %d мин.", text variable: PLC_PRG.mpx_s2_1_battery_time
    hotkey  Id=481037385728, Key=KeyDown=True, KeyName=0, VisuElemId=7
    hotkey  Id=481038434304, Key=KeyName=0, VisuElemId=7
END_VISUALIZATION

// CODESYS_Control_for_Raspberry_Pi/Application/visualization/test
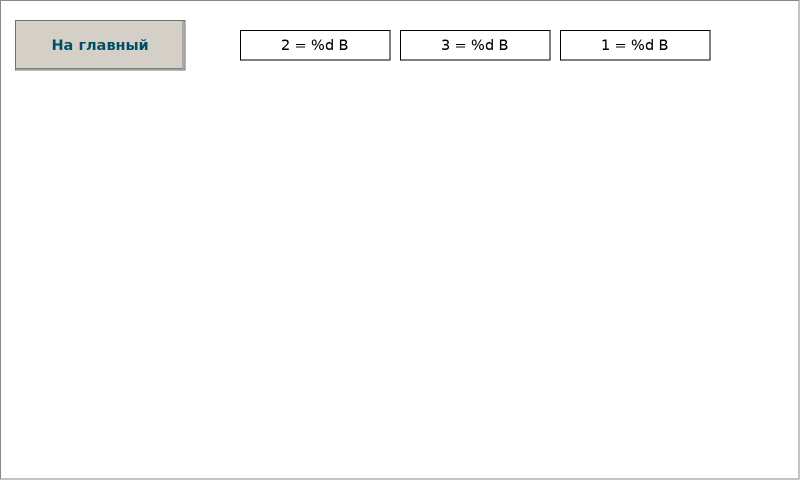
VISUALIZATION test  // 800x480, background image ImagePool.bg_800
    Button (15,20 170x50), "На главный"
        OnMouseClick:  Assign=main, Type=Assignment
    Rectangle (560,30 150x30), "1 = %d В", text variable: PLC_PRG.pot_1
    Rectangle (240,30 150x30), "2 = %d В", text variable: PLC_PRG.pot_2
    Rectangle (400,30 150x30), "3 = %d В", text variable: PLC_PRG.pot_3
    hotkey  Id=481037385728, Key=KeyDown=True, KeyName=0, VisuElemId=1
    hotkey  Id=481038434304, Key=KeyName=0, VisuElemId=1
END_VISUALIZATION

// CODESYS_Control_for_Raspberry_Pi/Application/visualization/ups_s2/ups_s2
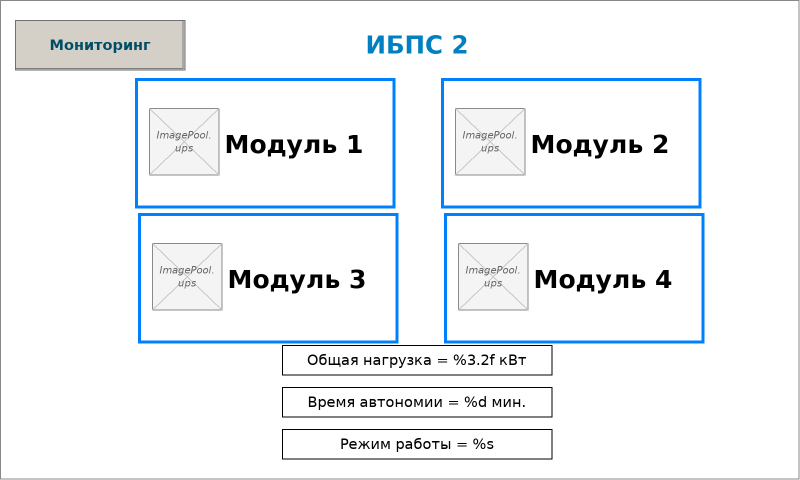
VISUALIZATION ups_s2  // 800x480, background image ImagePool.bg_800
    Rectangle (214,30 406x30), "ИБПС 2"
    Button (15,20 170x50), "Мониторинг"
        OnMouseClick:  Assign=monitoring, Type=Assignment
    Group (138,213 260x115)
        OnMouseClick:  Assign=ups_s2_m3_state, Type=Assignment
        RoundedRectangle (0,0 260x130), colour toggle: InterviewState.MPX_S1_3_State
        Image (14,30 70x67), image: ImagePool.ups
        RoundedRectangle (80,38 158x56), "Модуль 3"
            OnMouseClick:  Assign=ups_s2_m1_state, Type=Assignment
    Group (135,78 260x115)
        OnMouseClick:  Assign=ups_s2_m1_state, Type=Assignment
        RoundedRectangle (0,0 260x130), colour toggle: InterviewState.MPX_S1_1_State
        Image (14,30 70x67), image: ImagePool.ups
        RoundedRectangle (80,38 158x56), "Модуль 1"
            OnMouseClick:  Assign=ups_s2_m1_state, Type=Assignment
    Group (444,213 260x115)
        OnMouseClick:  Assign=ups_s2_m4_state, Type=Assignment
        RoundedRectangle (0,0 260x130), colour toggle: InterviewState.MPX_S1_4_State
        Image (14,30 70x67), image: ImagePool.ups
        RoundedRectangle (80,38 158x56), "Модуль 4"
            OnMouseClick:  Assign=ups_s2_m1_state, Type=Assignment
    Group (441,78 260x115)
        OnMouseClick:  Assign=ups_s2_m2_state, Type=Assignment
        RoundedRectangle (0,0 260x130), colour toggle: InterviewState.MPX_S1_2_State
        Image (14,30 70x67), image: ImagePool.ups
        RoundedRectangle (80,38 158x56), "Модуль 2"
            OnMouseClick:  Assign=ups_s2_m1_state, Type=Assignment
    Rectangle (282,345 270x30), "Общая нагрузка = %3.2f кВт", text variable: PLC_PRG.mpx_s2_all_power
    Rectangle (282,387 270x30), "Время автономии = %d мин.", text variable: PLC_PRG.mpx_s2_1_battery_time
    Rectangle (282,429 270x30), "Режим работы = %s", text variable: PLC_PRG.mpx_s2_state_string
    hotkey  Id=481037385728, Key=KeyDown=True, KeyName=0, VisuElemId=38
    hotkey  Id=481038434304, Key=KeyName=0, VisuElemId=38
END_VISUALIZATION

// CODESYS_Control_for_Raspberry_Pi/Application/visualization/main
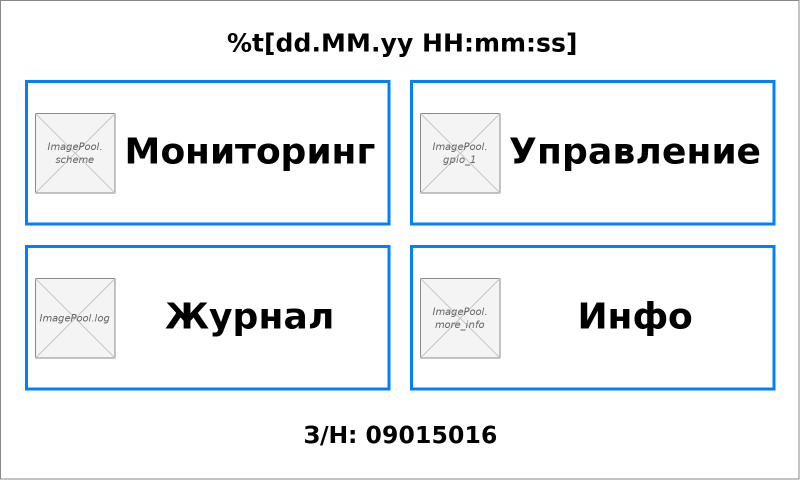
VISUALIZATION main  // 800x480, background image ImagePool.bg_800
    Group (25,80 365x145)
        OnMouseClick:  Assign=monitoring, Type=Assignment
        RoundedRectangle (0,0 365x145)
            OnMouseClick:  Assign=ups_s2_m1_state, Type=Assignment
        RoundedRectangle (95,43 260x56), "Мониторинг"
        Image (10,33 80x80), image: ImagePool.scheme
    Group (410,80 365x145)
        OnMouseClick:  Assign=control, Type=Assignment
        RoundedRectangle (0,0 365x145)
            OnMouseClick:  Assign=ups_s2_m1_state, Type=Assignment
        RoundedRectangle (95,43 260x56), "Управление"
            OnMouseClick:  Assign=ups_s2_m1_state, Type=Assignment
        Image (10,33 80x80), image: ImagePool.gpio_1
    Group (25,245 365x145)
        OnMouseClick:  Assign=logs, Type=Assignment
        RoundedRectangle (0,0 365x145)
            OnMouseClick:  Assign=ups_s2_m1_state, Type=Assignment
        RoundedRectangle (95,43 260x56), "Журнал"
            OnMouseClick:  Assign=ups_s2_m1_state, Type=Assignment
        Image (10,33 80x80), image: ImagePool.log
    Group (410,245 365x145)
        OnMouseClick:  Assign=more, Type=Assignment
        RoundedRectangle (0,0 365x145)
            OnMouseClick:  Assign=ups_s2_m1_state, Type=Assignment
        RoundedRectangle (95,43 260x56), "Инфо"
        Image (10,33 80x80), image: ImagePool.more_info
    Rectangle (215,20 375x45), "%t[dd.MM.yy HH:mm:ss]"
    Label (303,420 195x30), "З/Н: 09015016"
END_VISUALIZATION

// CODESYS_Control_for_Raspberry_Pi/Application/visualization/info
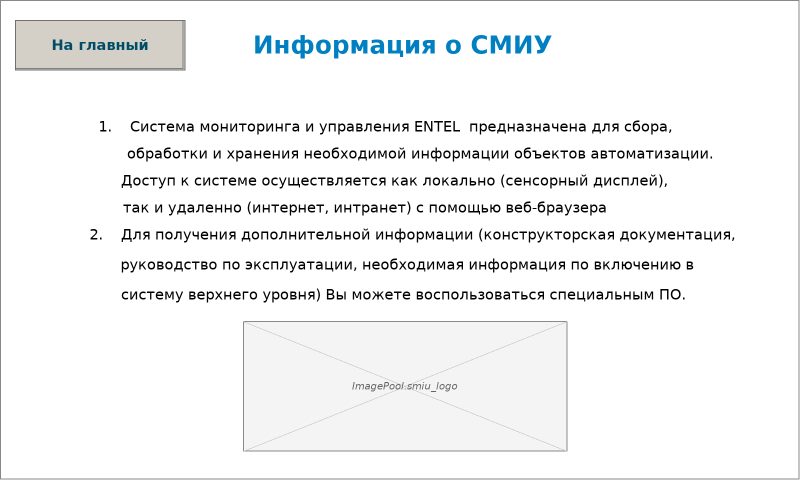
VISUALIZATION info  // 800x480, background image ImagePool.bg_800
    Rectangle (200,30 406x30), "Информация о СМИУ"
    Button (15,20 170x50), "На главный"
        OnMouseClick:  Assign=main, Type=Assignment
    Label (78,108 615x37), "1. Система мониторинга и управления ENTEL предназначена для сбора,"
    Label (120,135 601x37), "обработки и хранения необходимой информации объектов автоматизации."
    Label (99,162 591x37), "Доступ к системе осуществляется как локально (сенсорный дисплей),"
    Label (42,189 646x37), "так и удаленно (интернет, интранет) с помощью веб-браузера"
    Label (105,216 615x37), "2. Для получения дополнительной информации (конструкторская документация,"
    Label (120,243 601x37)
    Label (114,246 591x37), "руководство по эксплуатации, необходимая информация по включению в"
    Label (108,276 591x37), "систему верхнего уровня) Вы можете воспользоваться специальным ПО."
    Image (243,321 324x130), image: ImagePool.smiu_logo
END_VISUALIZATION

// CODESYS_Control_for_Raspberry_Pi/Application/visualization/climate
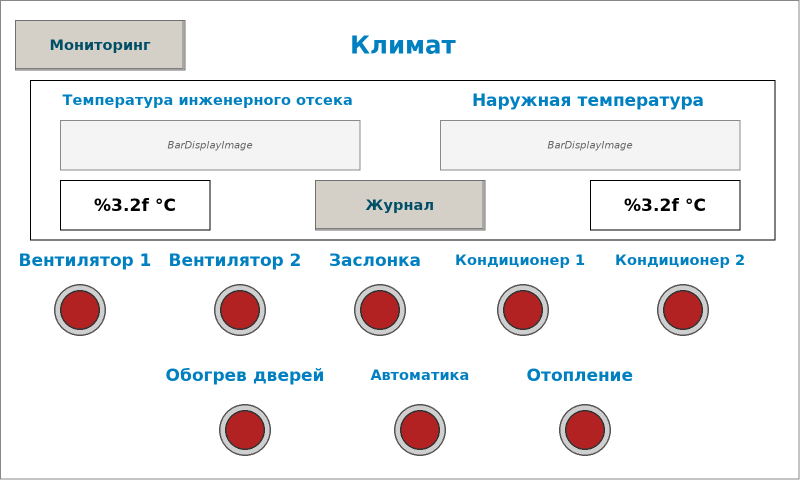
VISUALIZATION climate  // 800x480, background image ImagePool.bg_800
    Rectangle (200,30 406x30), "Климат"
    Button (15,20 170x50), "Мониторинг"
        OnMouseClick:  Assign=monitoring, Type=Assignment
    Rectangle (30,80 745x160)
    Rectangle (35,85 346x30), "Температура инженерного отсека"
    Rectangle (60,180 150x50), "%3.2f °С", text variable: PLC_PRG.climate_temp_in_real
    BarDisplayImage (60,120 300x50), value: PLC_PRG.climate_temp_in_real, style: BarDisplayImage-Gray, scale format: %.1f, scale -10..50
    Rectangle (415,85 346x30), "Наружная температура"
    Rectangle (590,180 150x50), "%3.2f °С", text variable: PLC_PRG.climate_temp_out_real
    BarDisplayImage (440,120 300x50), value: PLC_PRG.climate_temp_out_real, style: BarDisplayImage-Gray, scale format: %.1f, scale -60..80
    Rectangle (345,360 150x30), "Автоматика"
    Lamp1 (390,400 60x60), variable: PLC_PRG.climate_auto_state, style: Lamp-Lamp1-Red
    Lamp1 (50,280 60x60), variable: PLC_PRG.climate_vent_1_state, style: Lamp-Lamp1-Red
    Rectangle (10,250 150x20), "Вентилятор 1"
    Lamp1 (350,280 60x60), variable: PLC_PRG.climate_zaslonka_state, style: Lamp-Lamp1-Red
    Rectangle (320,250 110x20), "Заслонка"
    Rectangle (440,250 160x20), "Кондиционер 1"
    Lamp1 (490,280 66x60), variable: PLC_PRG.climate_condition_1_state, style: Lamp-Lamp1-Red
    Lamp1 (555,400 60x60), variable: PLC_PRG.climate_heat_state, style: Lamp-Lamp1-Red
    Rectangle (505,365 150x20), "Отопление"
    Lamp1 (210,280 60x60), variable: PLC_PRG.climate_vent_2_state, style: Lamp-Lamp1-Red
    Rectangle (160,250 150x20), "Вентилятор 2"
    Rectangle (600,250 160x20), "Кондиционер 2"
    Lamp1 (650,280 66x60), variable: PLC_PRG.climate_condition_2_state, style: Lamp-Lamp1-Red
    Lamp1 (215,400 60x60), variable: PLC_PRG.climate_heat_door_state, style: Lamp-Lamp1-Red
    Rectangle (155,365 180x20), "Обогрев дверей"
    Button (315,180 170x50), "Журнал"
        OnMouseClick:  Assign=climate_log, Type=Assignment
    hotkey  Id=481037385728, Key=KeyDown=True, KeyName=0, VisuElemId=3
    hotkey  Id=481038434304, Key=KeyName=0, VisuElemId=3
    hotkey  Id=481037385728, Key=KeyDown=True, KeyName=0, VisuElemId=73
    hotkey  Id=481038434304, Key=KeyName=0, VisuElemId=73
END_VISUALIZATION

// CODESYS_Control_for_Raspberry_Pi/Application/visualization/control
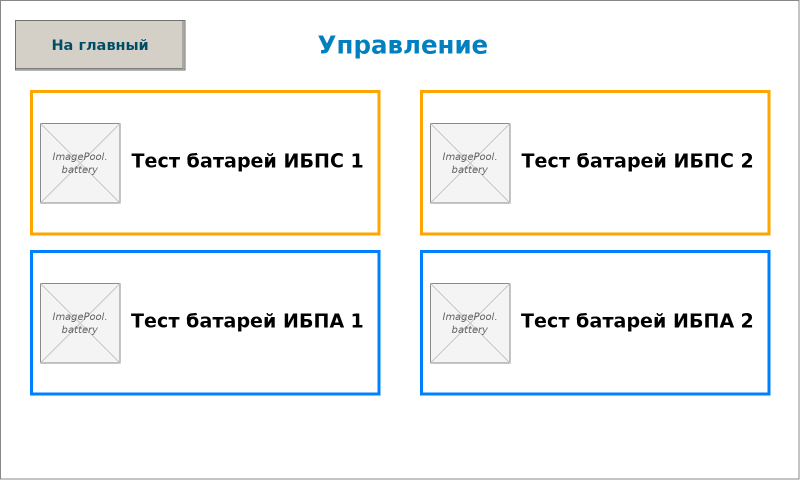
VISUALIZATION control  // 800x480, background image ImagePool.bg_800
    Rectangle (200,30 406x30), "Управление"
    Button (15,20 170x50), "На главный"
        OnMouseClick:  Assign=main, Type=Assignment
    Group (30,90 350x145)
        OnMouseClick:  ToggleVariable=PLC_PRG.mpx_s1_test_battery_start
        RoundedRectangle (0,0 350x145)
        RoundedRectangle (95,43 245x56), "Тест батарей ИБПС 1"
        Image (10,33 80x80), image: ImagePool.battery
    Group (420,90 350x145)
        OnMouseClick:  ToggleVariable=PLC_PRG.mpx_s2_test_battery_start
        RoundedRectangle (0,0 350x145)
            OnMouseClick:  ToggleVariable=PLC_PRG.mpx_s2_test_battery_start
        RoundedRectangle (95,43 245x56), "Тест батарей ИБПС 2"
        Image (10,33 80x80), image: ImagePool.battery
    Group (420,250 350x145)
        OnMouseClick:  ToggleVariable=PLC_PRG.mpx_a2_test_battery_start
        RoundedRectangle (0,0 350x145)
        RoundedRectangle (95,43 245x56), "Тест батарей ИБПА 2"
        Image (10,33 80x80), image: ImagePool.battery
    Group (30,250 350x145)
        OnMouseClick:  ToggleVariable=PLC_PRG.mpx_a1_test_battery_start
        RoundedRectangle (0,0 350x145)
        RoundedRectangle (95,43 245x56), "Тест батарей ИБПА 1"
        Image (10,33 80x80), image: ImagePool.battery
    hotkey  Id=481037385728, Key=KeyDown=True, KeyName=0, VisuElemId=3
    hotkey  Id=481038434304, Key=KeyName=0, VisuElemId=3
END_VISUALIZATION

// CODESYS_Control_for_Raspberry_Pi/Application/visualization/alarm
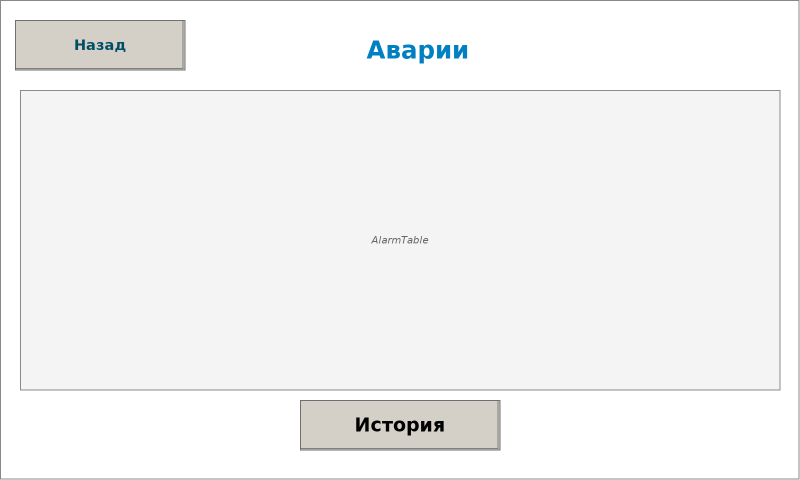
VISUALIZATION alarm  // 800x480, background image ImagePool.bg_800
    Button (300,400 200x50), "История", colour toggle: PLC_PRG.history
        toggle PLC_PRG.history
    Button (15,20 170x50), "Назад"
        OnMouseClick:  Assign=monitoring, Type=Previous
    AlarmTable (20,90 760x300)
        Column[0]: ColumnTitle=Временная отметка
        Column[1]: ColumnTitle=Сообщение
        p1521930926: AlarmGroup
        p1663851261: __All
        p3266827225: PLC_PRG.history
    Rectangle (215,35 406x30), "Аварии"
    hotkey  Id=481037385728, Key=KeyDown=True, KeyName=0, VisuElemId=6
    hotkey  Id=481038434304, Key=KeyName=0, VisuElemId=6
END_VISUALIZATION

// CODESYS_Control_for_Raspberry_Pi/Application/visualization/schrps
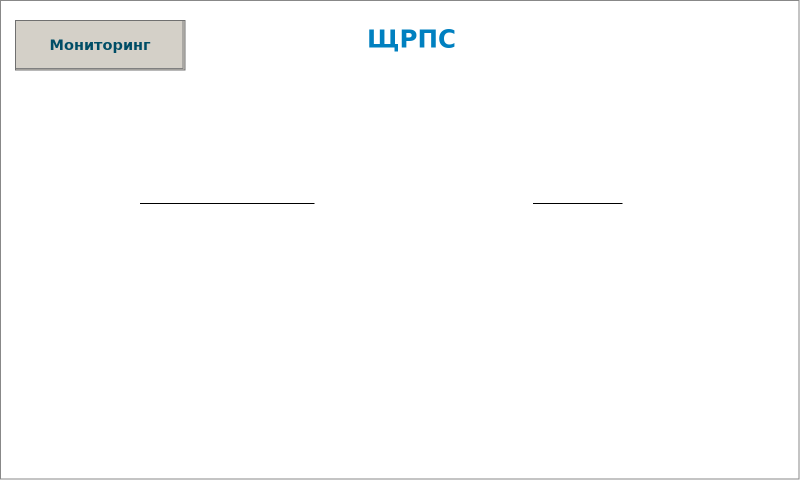
VISUALIZATION schrps  // 800x480, background image ImagePool.schrps
    Button (15,20 170x50), "Мониторинг"
        OnMouseClick:  Assign=monitoring, Type=Assignment
    Line (140,203) (314,203), colour toggle: NOT(PLC_PRG.mv110_in_7_gp1_u_fault)
    Line (533,203) (622,203), colour toggle: NOT(PLC_PRG.mv110_in_8_gp2_u_fault)
    Rectangle (316,24 191x30), "ЩРПC"
    hotkey  Id=481037385728, Key=KeyDown=True, KeyName=0, VisuElemId=1
    hotkey  Id=481038434304, Key=KeyName=0, VisuElemId=1
END_VISUALIZATION

// CODESYS_Control_for_Raspberry_Pi/Application/visualization/shasn
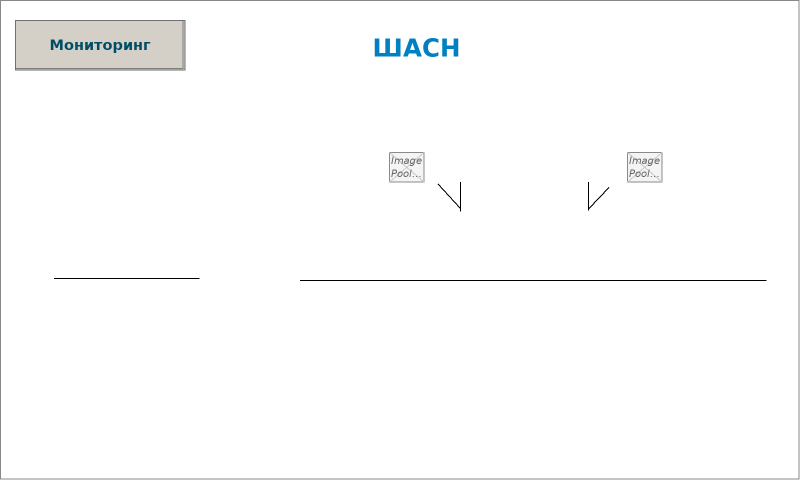
VISUALIZATION shasn  // 800x480, background image ImagePool.shasn
    Button (15,20 170x50), "Мониторинг"
        OnMouseClick:  Assign=monitoring, Type=Assignment
    Line (426,184)
    Line (460,208) (438,184), invisible if: PLC_PRG.mv110_in_4_qs1_1position
    Line (460,182) (460,211), invisible if: NOT(PLC_PRG.mv110_in_4_qs1_1position)
    Line (589,208) (609,187), invisible if: PLC_PRG.mv110_in_5_qs1_2position
    Line (588,182) (588,210), invisible if: NOT(PLC_PRG.mv110_in_5_qs1_2position)
    Line (300,280) (766,280), colour toggle: PLC_PRG.mv110_in_3_gp_sn_present
    Line (54,278) (199,278), colour toggle: PLC_PRG.mv110_in_2_bp_sn_present
    Image (389,152 35x30), invisible if: NOT(PLC_PRG.mv110_in_0_in_main_present), image: ImagePool.volt
    Line (664,184)
    Image (627,152 35x30), invisible if: NOT(PLC_PRG.mv110_in_1_in_reserve_present), image: ImagePool.volt
    Rectangle (321,33 191x30), "ШАСН"
    hotkey  Id=481037385728, Key=KeyDown=True, KeyName=0, VisuElemId=1
    hotkey  Id=481038434304, Key=KeyName=0, VisuElemId=1
END_VISUALIZATION

// CODESYS_Control_for_Raspberry_Pi/Application/visualization/logs
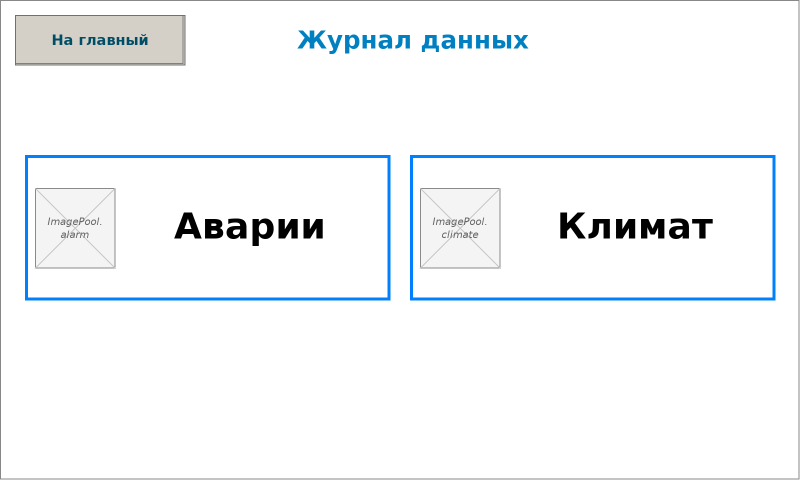
VISUALIZATION logs  // 800x480, background image ImagePool.bg_800
    Button (15,15 170x50), "На главный"
        OnMouseClick:  Assign=main, Type=Assignment
    Rectangle (210,25 406x30), "Журнал данных"
    Group (25,155 365x145)
        OnMouseClick:  Assign=alarm, Type=Assignment
        RoundedRectangle (0,0 365x145)
            OnMouseClick:  Assign=ups_s2_m1_state, Type=Assignment
        RoundedRectangle (95,43 260x56), "Аварии"
        Image (10,33 80x80), image: ImagePool.alarm
    Group (410,155 365x145)
        OnMouseClick:  Assign=climate_log, Type=Assignment
        RoundedRectangle (0,0 365x145)
            OnMouseClick:  Assign=ups_s2_m1_state, Type=Assignment
        RoundedRectangle (95,43 260x56), "Климат"
        Image (10,33 80x80), image: ImagePool.climate
    hotkey  Id=481037385728, Key=KeyDown=True, KeyName=0, VisuElemId=1
    hotkey  Id=481038434304, Key=KeyName=0, VisuElemId=1
END_VISUALIZATION

// CODESYS_Control_for_Raspberry_Pi/Application/visualization/schrpa
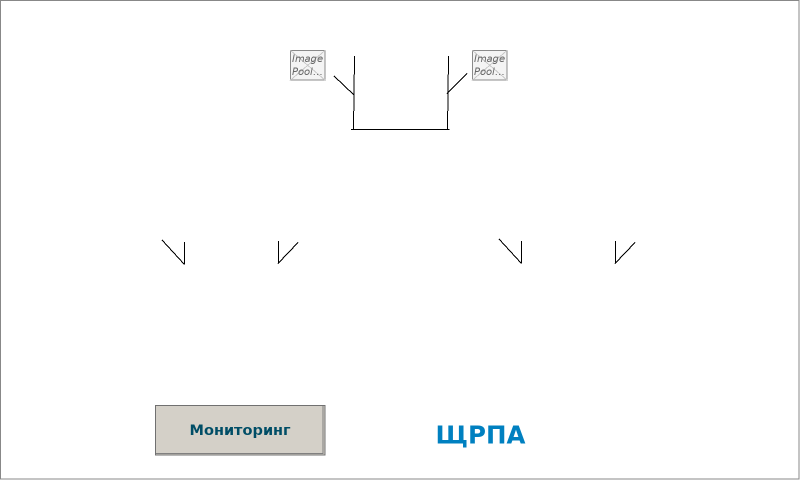
VISUALIZATION schrpa  // 800x480, background image ImagePool.schrpa
    Button (155,405 170x50), "Мониторинг"
        OnMouseClick:  Assign=monitoring, Type=Assignment
    Rectangle (385,420 191x30), "ЩРПА"
    Image (290,50 35x30), invisible if: NOT(GPIO_HANDLER.IN_4), image: ImagePool.volt
    Image (472,50 35x30), invisible if: NOT(GPIO_HANDLER.IN_5), image: ImagePool.volt
    Line (354,56) (353,129), invisible if: NOT(GPIO_HANDLER.IN_6)
    Line (354,95) (334,76), invisible if: GPIO_HANDLER.IN_6
    Line (351,129) (400,129), invisible if: NOT(GPIO_HANDLER.IN_6)
    Line (447,93) (467,73), invisible if: GPIO_HANDLER.IN_7
    Line (448,56) (447,129), invisible if: NOT(GPIO_HANDLER.IN_7)
    Line (400,129) (449,129), invisible if: NOT(GPIO_HANDLER.IN_7)
    Line (150,240)
    Line (184,264) (162,240), invisible if: GPIO_HANDLER.IN_8
    Line (184,242) (184,264), invisible if: NOT(GPIO_HANDLER.IN_8)
    Line (278,263) (298,242), invisible if: GPIO_HANDLER.IN_9
    Line (278,241) (278,263), invisible if: NOT(GPIO_HANDLER.IN_9)
    Line (487,239)
    Line (521,263) (499,239), invisible if: GPIO_HANDLER.IN_11
    Line (521,241) (521,263), invisible if: NOT(GPIO_HANDLER.IN_11)
    Line (615,263) (635,242), invisible if: GPIO_HANDLER.IN_10
    Line (615,241) (615,263), invisible if: NOT(GPIO_HANDLER.IN_10)
    hotkey  Id=481037385728, Key=KeyDown=True, KeyName=0, VisuElemId=1
    hotkey  Id=481038434304, Key=KeyName=0, VisuElemId=1
END_VISUALIZATION

// CODESYS_Control_for_Raspberry_Pi/Application/visualization/ups_s2/ups_s2_m2_params
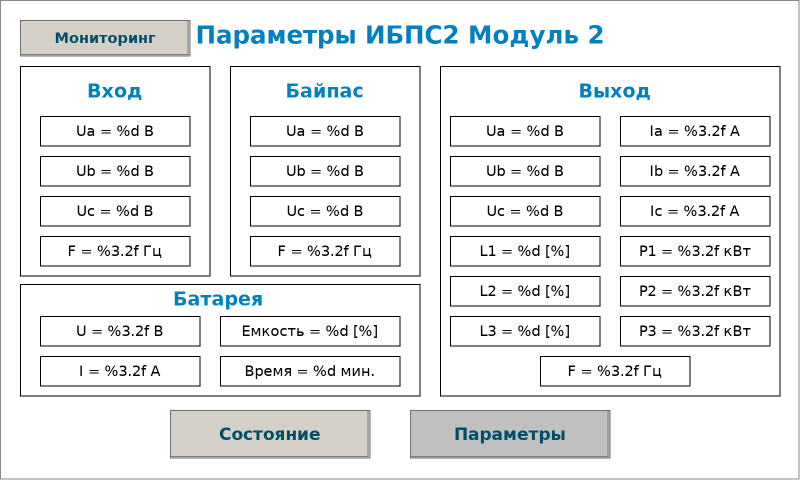
VISUALIZATION ups_s2_m2_params  // 800x480, background image ImagePool.bg_800
    Rectangle (186,20 428x30), "Параметры ИБПC2 Модуль 2"
    Button (170,410 200x48), "Состояние"
        OnMouseClick:  Assign=ups_s2_m2_state, Type=Assignment
    Button (410,410 200x48), "Параметры", pressed state: PLC_PRG.var_true
    Button (20,20 170x36), "Мониторинг"
        OnMouseClick:  Assign=monitoring, Type=Assignment
    Rectangle (20,66 190x210)
    Rectangle (440,66 340x330)
    Rectangle (30,76 170x30), "Вход"
    Rectangle (40,116 150x30), "Ua = %d В", text variable: PLC_PRG.mpx_s2_2_in_v_1
    Rectangle (40,156 150x30), "Ub = %d В", text variable: PLC_PRG.mpx_s2_2_in_v_2
    Rectangle (40,196 150x30), "Uc = %d В", text variable: PLC_PRG.mpx_s2_2_in_v_3
    Rectangle (40,236 150x30), "F = %3.2f Гц", text variable: PLC_PRG.mpx_s2_2_in_freq_real
    Rectangle (230,66 190x210)
    Rectangle (240,76 170x30), "Байпас"
    Rectangle (250,116 150x30), "Ua = %d В", text variable: PLC_PRG.mpx_s2_2_bypass_v_1
    Rectangle (250,156 150x30), "Ub = %d В", text variable: PLC_PRG.mpx_s2_2_bypass_v_2
    Rectangle (250,196 150x30), "Uc = %d В", text variable: PLC_PRG.mpx_s2_2_bypass_v_3
    Rectangle (250,236 150x30), "F = %3.2f Гц", text variable: PLC_PRG.mpx_s2_2_bypass_freq_real
    Rectangle (460,76 310x30), "Выход"
    Rectangle (450,116 150x30), "Ua = %d В", text variable: PLC_PRG.mpx_s2_2_output_v_1
    Rectangle (450,156 150x30), "Ub = %d В", text variable: PLC_PRG.mpx_s2_2_output_v_2
    Rectangle (450,196 150x30), "Uc = %d В", text variable: PLC_PRG.mpx_s2_2_output_v_3
    Rectangle (620,116 150x30), "Ia = %3.2f A", text variable: PLC_PRG.mpx_s2_2_output_i_1_real
    Rectangle (620,156 150x30), "Ib = %3.2f A", text variable: PLC_PRG.mpx_s2_2_output_i_2_real
    Rectangle (620,196 150x30), "Ic = %3.2f A", text variable: PLC_PRG.mpx_s2_2_output_i_3_real
    Rectangle (450,236 150x30), "L1 = %d [%]", text variable: PLC_PRG.mpx_s2_2_load_ph_1
    Rectangle (450,276 150x30), "L2 = %d [%]", text variable: PLC_PRG.mpx_s2_2_load_ph_2
    Rectangle (450,316 150x30), "L3 = %d [%]", text variable: PLC_PRG.mpx_s2_2_load_ph_3
    Rectangle (620,236 150x30), "P1 = %3.2f кВт", text variable: PLC_PRG.mpx_s2_2_output_active_power_1_real
    Rectangle (620,276 150x30), "P2 = %3.2f кВт", text variable: PLC_PRG.mpx_s2_2_output_active_power_2_real
    Rectangle (620,316 150x30), "P3 = %3.2f кВт", text variable: PLC_PRG.mpx_s2_2_output_active_power_3_real
    Rectangle (540,356 150x30), "F = %3.2f Гц", text variable: PLC_PRG.mpx_s2_2_output_freq_real
    Rectangle (20,284 400x112)
    Rectangle (30,290 376x18), "Батарея"
    Rectangle (40,316 160x30), "U = %3.2f В", text variable: PLC_PRG.mpx_s2_2_battery_voltage_real
    Rectangle (40,356 160x30), "I = %3.2f A", text variable: PLC_PRG.mpx_s2_2_battery_current_real
    Rectangle (220,316 180x30), "Емкость = %d [%]", text variable: PLC_PRG.mpx_s2_2_battery_capacity
    Rectangle (220,356 180x30), "Время = %d мин.", text variable: PLC_PRG.mpx_s2_2_battery_time
    hotkey  Id=481037385728, Key=KeyDown=True, KeyName=0, VisuElemId=7
    hotkey  Id=481038434304, Key=KeyName=0, VisuElemId=7
END_VISUALIZATION

// CODESYS_Control_for_Raspberry_Pi/Application/visualization/ups_s2/ups_s2_m2_state
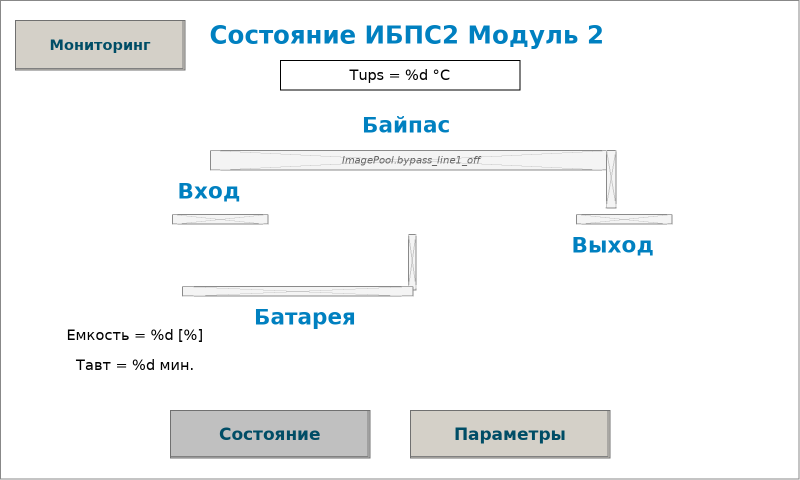
VISUALIZATION ups_s2_m2_state  // 800x480, background image ImagePool.mpx_state_bg
    Rectangle (204,20 406x30), "Состояние ИБПС2 Модуль 2"
    Button (410,410 200x48), "Параметры"
        OnMouseClick:  Assign=ups_s2_m2_params, Type=Assignment
    Button (170,410 200x48), "Состояние", pressed state: PLC_PRG.var_true
    Rectangle (350,110 112x30), "Байпас"
    Rectangle (246,302 118x30), "Батарея"
    Rectangle (166,176 86x30), "Вход"
    Rectangle (560,230 106x30), "Выход"
    Rectangle (280,60 240x30), "Tups = %d °С", text variable: PLC_PRG.mpx_s2_2_temp
    Rectangle (30,320 210x30), "Емкость = %d [%]", text variable: PLC_PRG.mpx_s2_2_battery_capacity
    Rectangle (30,350 210x30), "Tавт = %d мин.", text variable: PLC_PRG.mpx_s2_2_battery_time
    Image (210,150 402x20), image: ImagePool.bypass_line1_off
        p84334746: PLC_PRG.mpx_s2_2_bypass_line_state
    Image (606,150 10x58), image: ImagePool.bypass_arrow_off
        p84334746: PLC_PRG.mpx_s2_2_bypass_arrow_state
    Image (576,214 96x10), image: ImagePool.arrow_off
        p84334746: PLC_PRG.mpx_s2_2_output_state
    Image (172,214 96x10), image: ImagePool.arrow_off
        p84334746: PLC_PRG.mpx_s2_2_input_state
    Image (408,234 8x56), image: ImagePool.battery_arrow_off
        p84334746: PLC_PRG.mpx_s2_2_battery_arrow_state
    Image (182,286 231x10), image: ImagePool.battery_line_off
        p84334746: PLC_PRG.mpx_s2_2_battery_line_state
    Button (15,20 170x50), "Мониторинг"
        OnMouseClick:  Assign=monitoring, Type=Assignment
    hotkey  Id=481037385728, Key=KeyDown=True, KeyName=0, VisuElemId=38
    hotkey  Id=481038434304, Key=KeyName=0, VisuElemId=38
END_VISUALIZATION

// CODESYS_Control_for_Raspberry_Pi/Application/visualization/ups_s2/ups_s2_m3_params
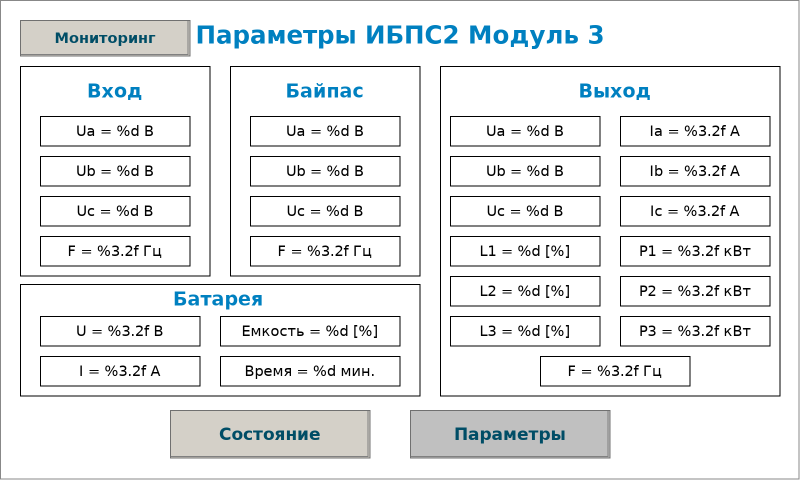
VISUALIZATION ups_s2_m3_params  // 800x480, background image ImagePool.bg_800
    Rectangle (186,20 428x30), "Параметры ИБПC2 Модуль 3"
    Button (170,410 200x48), "Состояние"
        OnMouseClick:  Assign=ups_s2_m3_state, Type=Assignment
    Button (410,410 200x48), "Параметры", pressed state: PLC_PRG.var_true
    Button (20,20 170x36), "Мониторинг"
        OnMouseClick:  Assign=monitoring, Type=Assignment
    Rectangle (20,66 190x210)
    Rectangle (440,66 340x330)
    Rectangle (30,76 170x30), "Вход"
    Rectangle (40,116 150x30), "Ua = %d В", text variable: PLC_PRG.mpx_s2_3_in_v_1
    Rectangle (40,156 150x30), "Ub = %d В", text variable: PLC_PRG.mpx_s2_3_in_v_2
    Rectangle (40,196 150x30), "Uc = %d В", text variable: PLC_PRG.mpx_s2_3_in_v_3
    Rectangle (40,236 150x30), "F = %3.2f Гц", text variable: PLC_PRG.mpx_s2_3_in_freq_real
    Rectangle (230,66 190x210)
    Rectangle (240,76 170x30), "Байпас"
    Rectangle (250,116 150x30), "Ua = %d В", text variable: PLC_PRG.mpx_s2_3_bypass_v_1
    Rectangle (250,156 150x30), "Ub = %d В", text variable: PLC_PRG.mpx_s2_3_bypass_v_2
    Rectangle (250,196 150x30), "Uc = %d В", text variable: PLC_PRG.mpx_s2_3_bypass_v_3
    Rectangle (250,236 150x30), "F = %3.2f Гц", text variable: PLC_PRG.mpx_s2_3_bypass_freq_real
    Rectangle (460,76 310x30), "Выход"
    Rectangle (450,116 150x30), "Ua = %d В", text variable: PLC_PRG.mpx_s2_3_output_v_1
    Rectangle (450,156 150x30), "Ub = %d В", text variable: PLC_PRG.mpx_s2_3_output_v_2
    Rectangle (450,196 150x30), "Uc = %d В", text variable: PLC_PRG.mpx_s2_3_output_v_3
    Rectangle (620,116 150x30), "Ia = %3.2f A", text variable: PLC_PRG.mpx_s2_3_output_i_1_real
    Rectangle (620,156 150x30), "Ib = %3.2f A", text variable: PLC_PRG.mpx_s2_3_output_i_2_real
    Rectangle (620,196 150x30), "Ic = %3.2f A", text variable: PLC_PRG.mpx_s2_3_output_i_3_real
    Rectangle (450,236 150x30), "L1 = %d [%]", text variable: PLC_PRG.mpx_s2_3_load_ph_1
    Rectangle (450,276 150x30), "L2 = %d [%]", text variable: PLC_PRG.mpx_s2_3_load_ph_2
    Rectangle (450,316 150x30), "L3 = %d [%]", text variable: PLC_PRG.mpx_s2_3_load_ph_3
    Rectangle (620,236 150x30), "P1 = %3.2f кВт", text variable: PLC_PRG.mpx_s2_3_output_active_power_1_real
    Rectangle (620,276 150x30), "P2 = %3.2f кВт", text variable: PLC_PRG.mpx_s2_3_output_active_power_2_real
    Rectangle (620,316 150x30), "P3 = %3.2f кВт", text variable: PLC_PRG.mpx_s2_3_output_active_power_3_real
    Rectangle (540,356 150x30), "F = %3.2f Гц", text variable: PLC_PRG.mpx_s2_3_output_freq_real
    Rectangle (20,284 400x112)
    Rectangle (30,290 376x18), "Батарея"
    Rectangle (40,316 160x30), "U = %3.2f В", text variable: PLC_PRG.mpx_s2_3_battery_voltage_real
    Rectangle (40,356 160x30), "I = %3.2f A", text variable: PLC_PRG.mpx_s2_3_battery_current_real
    Rectangle (220,316 180x30), "Емкость = %d [%]", text variable: PLC_PRG.mpx_s2_3_battery_capacity
    Rectangle (220,356 180x30), "Время = %d мин.", text variable: PLC_PRG.mpx_s2_3_battery_time
    hotkey  Id=481037385728, Key=KeyDown=True, KeyName=0, VisuElemId=7
    hotkey  Id=481038434304, Key=KeyName=0, VisuElemId=7
END_VISUALIZATION

// CODESYS_Control_for_Raspberry_Pi/Application/visualization/ups_s2/ups_s2_m4_state
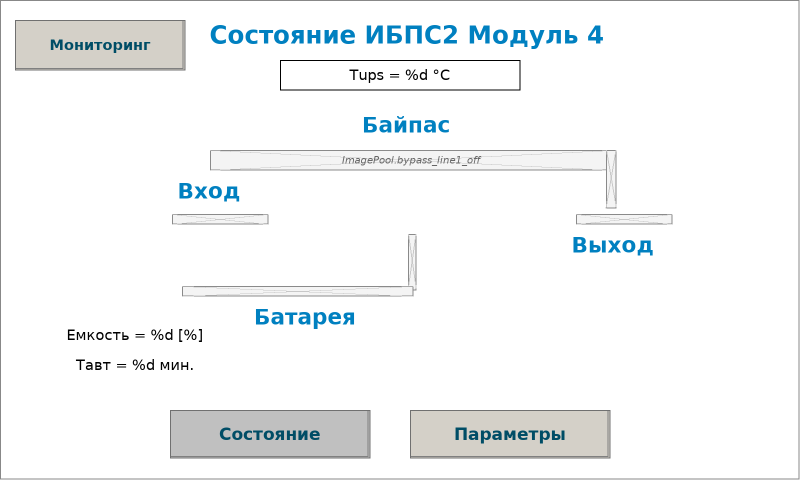
VISUALIZATION ups_s2_m4_state  // 800x480, background image ImagePool.mpx_state_bg
    Rectangle (204,20 406x30), "Состояние ИБПС2 Модуль 4"
    Button (410,410 200x48), "Параметры"
        OnMouseClick:  Assign=ups_s2_m4_params, Type=Assignment
    Button (170,410 200x48), "Состояние", pressed state: PLC_PRG.var_true
    Rectangle (350,110 112x30), "Байпас"
    Rectangle (246,302 118x30), "Батарея"
    Rectangle (166,176 86x30), "Вход"
    Rectangle (560,230 106x30), "Выход"
    Rectangle (280,60 240x30), "Tups = %d °С", text variable: PLC_PRG.mpx_s2_4_temp
    Rectangle (30,320 210x30), "Емкость = %d [%]", text variable: PLC_PRG.mpx_s2_4_battery_capacity
    Rectangle (30,350 210x30), "Tавт = %d мин.", text variable: PLC_PRG.mpx_s2_4_battery_time
    Image (210,150 402x20), image: ImagePool.bypass_line1_off
        p84334746: PLC_PRG.mpx_s2_4_bypass_line_state
    Image (606,150 10x58), image: ImagePool.bypass_arrow_off
        p84334746: PLC_PRG.mpx_s2_4_bypass_arrow_state
    Image (576,214 96x10), image: ImagePool.arrow_off
        p84334746: PLC_PRG.mpx_s2_4_output_state
    Image (172,214 96x10), image: ImagePool.arrow_off
        p84334746: PLC_PRG.mpx_s2_4_input_state
    Image (408,234 8x56), image: ImagePool.battery_arrow_off
        p84334746: PLC_PRG.mpx_s2_4_battery_arrow_state
    Image (182,286 231x10), image: ImagePool.battery_line_off
        p84334746: PLC_PRG.mpx_s2_4_battery_line_state
    Button (15,20 170x50), "Мониторинг"
        OnMouseClick:  Assign=monitoring, Type=Assignment
    hotkey  Id=481037385728, Key=KeyDown=True, KeyName=0, VisuElemId=38
    hotkey  Id=481038434304, Key=KeyName=0, VisuElemId=38
END_VISUALIZATION

// CODESYS_Control_for_Raspberry_Pi/Application/visualization/ups_s2/ups_s2_m4_params
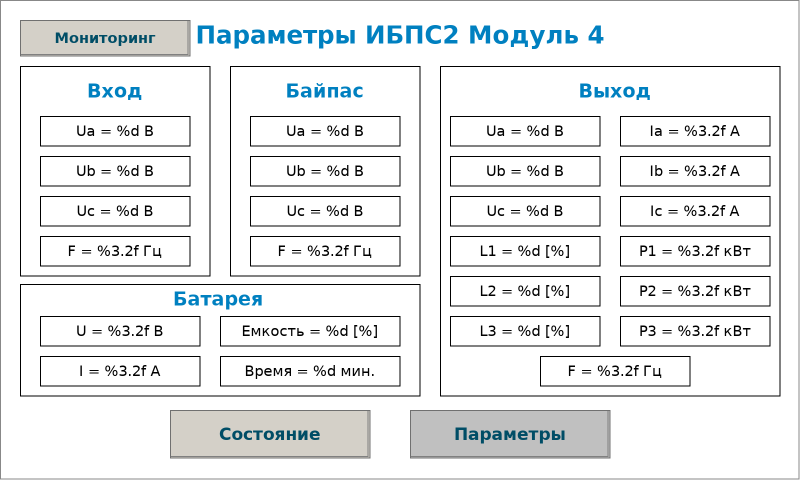
VISUALIZATION ups_s2_m4_params  // 800x480, background image ImagePool.bg_800
    Rectangle (186,20 428x30), "Параметры ИБПC2 Модуль 4"
    Button (170,410 200x48), "Состояние"
        OnMouseClick:  Assign=ups_s2_m4_state, Type=Assignment
    Button (410,410 200x48), "Параметры", pressed state: PLC_PRG.var_true
    Button (20,20 170x36), "Мониторинг"
        OnMouseClick:  Assign=monitoring, Type=Assignment
    Rectangle (20,66 190x210)
    Rectangle (440,66 340x330)
    Rectangle (30,76 170x30), "Вход"
    Rectangle (40,116 150x30), "Ua = %d В", text variable: PLC_PRG.mpx_s2_4_in_v_1
    Rectangle (40,156 150x30), "Ub = %d В", text variable: PLC_PRG.mpx_s2_4_in_v_2
    Rectangle (40,196 150x30), "Uc = %d В", text variable: PLC_PRG.mpx_s2_4_in_v_3
    Rectangle (40,236 150x30), "F = %3.2f Гц", text variable: PLC_PRG.mpx_s2_4_in_freq_real
    Rectangle (230,66 190x210)
    Rectangle (240,76 170x30), "Байпас"
    Rectangle (250,116 150x30), "Ua = %d В", text variable: PLC_PRG.mpx_s2_4_bypass_v_1
    Rectangle (250,156 150x30), "Ub = %d В", text variable: PLC_PRG.mpx_s2_4_bypass_v_2
    Rectangle (250,196 150x30), "Uc = %d В", text variable: PLC_PRG.mpx_s2_4_bypass_v_3
    Rectangle (250,236 150x30), "F = %3.2f Гц", text variable: PLC_PRG.mpx_s2_4_bypass_freq_real
    Rectangle (460,76 310x30), "Выход"
    Rectangle (450,116 150x30), "Ua = %d В", text variable: PLC_PRG.mpx_s2_4_output_v_1
    Rectangle (450,156 150x30), "Ub = %d В", text variable: PLC_PRG.mpx_s2_4_output_v_2
    Rectangle (450,196 150x30), "Uc = %d В", text variable: PLC_PRG.mpx_s2_4_output_v_3
    Rectangle (620,116 150x30), "Ia = %3.2f A", text variable: PLC_PRG.mpx_s2_4_output_i_1_real
    Rectangle (620,156 150x30), "Ib = %3.2f A", text variable: PLC_PRG.mpx_s2_4_output_i_2_real
    Rectangle (620,196 150x30), "Ic = %3.2f A", text variable: PLC_PRG.mpx_s2_4_output_i_3_real
    Rectangle (450,236 150x30), "L1 = %d [%]", text variable: PLC_PRG.mpx_s2_4_load_ph_1
    Rectangle (450,276 150x30), "L2 = %d [%]", text variable: PLC_PRG.mpx_s2_4_load_ph_2
    Rectangle (450,316 150x30), "L3 = %d [%]", text variable: PLC_PRG.mpx_s2_4_load_ph_3
    Rectangle (620,236 150x30), "P1 = %3.2f кВт", text variable: PLC_PRG.mpx_s2_4_output_active_power_1_real
    Rectangle (620,276 150x30), "P2 = %3.2f кВт", text variable: PLC_PRG.mpx_s2_4_output_active_power_2_real
    Rectangle (620,316 150x30), "P3 = %3.2f кВт", text variable: PLC_PRG.mpx_s2_4_output_active_power_3_real
    Rectangle (540,356 150x30), "F = %3.2f Гц", text variable: PLC_PRG.mpx_s2_4_output_freq_real
    Rectangle (20,284 400x112)
    Rectangle (30,290 376x18), "Батарея"
    Rectangle (40,316 160x30), "U = %3.2f В", text variable: PLC_PRG.mpx_s2_4_battery_voltage_real
    Rectangle (40,356 160x30), "I = %3.2f A", text variable: PLC_PRG.mpx_s2_4_battery_current_real
    Rectangle (220,316 180x30), "Емкость = %d [%]", text variable: PLC_PRG.mpx_s2_4_battery_capacity
    Rectangle (220,356 180x30), "Время = %d мин.", text variable: PLC_PRG.mpx_s2_4_battery_time
    hotkey  Id=481037385728, Key=KeyDown=True, KeyName=0, VisuElemId=7
    hotkey  Id=481038434304, Key=KeyName=0, VisuElemId=7
END_VISUALIZATION

